// ---- POUs/HAWinoCore/MQTT.TcPOU
PROGRAM MQTT
VAR
// Local Variables for Mqtt Client handling
	fbIotMqttClient : FB_IotMqttClient;
	bSetParameter 	: BOOL := TRUE;
	bConnect 		: BOOL := TRUE;	
	
// Publish message
	initMQTT : BOOL := FALSE;
	sTopicPubToPowerMgmt : STRING(255); //:= CONCAT('Robots/PowerMgmt/Robot_', INT_TO_STRING(.Var_HAWIno.Robot_Number)); 	// ToDo: Bisher ist die Nummer des HAWino fest kodiert
	sTopicPubToPowerMgmt_SOC : STRING(255);// := CONCAT('Robots/PowerMgmt/SoC_Robot_', INT_TO_STRING(.Var_HAWIno.Robot_Number)); 
	sPayloadPub : STRING(2000);	
	fbTimerPub 	: TON := (PT:=T#500MS);									// Intervall für das Senden des Akku-Status
	
//Received message
	bSubscribed    : BOOL;
	sTopicSubToPowerMgmt : STRING(255);// := CONCAT('PowerMgmt/Robots/Robot_', INT_TO_STRING(.Var_HAWIno.Robot_Number));	// ToDo: Bisher ist die Nummer des HAWino fest kodiert
	sTopicRcv      : STRING(255);
	sPayloadRcv    : STRING(255);
	sPayloadRcv_Status    : STRING(255);
	sPayloadRcv_Status_Test: STRING(255);
	fbMessageQueue : FB_IotMqttMessageQueue;
    fbMessage      : FB_IotMqttMessage;
	hrErrorOccurred : HRESULT; 			// Enthlt dern letzten augetretenen Fehler
	
//subscribe
	sTopicSubToGW1_Status : STRING(255);
	sTopicSubToGW1_Auftrag : STRING(255);
	sTopicSubCollision : STRING(255);
	sTopicPubCollision : ARRAY[1..4] OF STRING(255);
	sTopicSubReset : STRING(255);
	
// Variables for JSON
	fbJson			: FB_JsonSaxWriter;
	fbJsonDataType 	: FB_JsonReadWriteDataType;
	sJsonDoc       	: STRING(2000); 
	
// Local Variables for TwinCAT IoT Communication (TF6701) with direct link to EK1200 and TcCom
	//stMqtt_HAWino_In	AT%I*	: ST_PwrMgmt_HAWino_In;		// Attention! Don't link TIME Variables, otherwise we get an error!
	//stMqtt_HAWino_Out	AT%Q*	: ST_PwrMgmt_HAWino_Out;
	
	stMqtt_HAWino_In	 AT%I*: ST_PwrMgmt_HAWino_In;		// Attention! Don't link TIME Variables, otherwise we get an error!
	stMqtt_HAWino_Out	 AT%Q*: ST_PwrMgmt_HAWino_Out;
	
	SOC_Out : STRING(255);
	nBatteryTemperature	AT%I*	: INT;
	
	bComCheckAnswer	AT%Q*	: BOOL;
	
	stMqtt_HAWinoValues	: ST_PwrMgmt_HAWino;
	
	
// Timer to create a time stamp
	fbTimerTimestamp : TON := (PT:=T#71582M47S295MS);
	
// Local Vaiables to evaluate and act to input
	fbComCheckFlag	: RS;
	
	sTopicSubToFleetMgmt: STRING;
	Reset1: BOOL;
	//Input synccheck. robotdata has been read and can be used.
	txtReadInit AT%I* : BOOL := FALSE;
	
	//eigene Topics und Payload
	sTopicPubToGW1 : STRING(255);
	WerkstueckAusgelesen: BOOL;
	sPayloadPub1 : STRING(2000);
	Robotstatus : RobotStatusGW1;
	sTopicSubToGW1: STRING(255);
	nPayloadSize:INT;
	sPayloadPubCollision : STRING(100);
	n: INT;												
	
	FeedbackToGW1 AT%I*: STRING(50);				//Statusmeldungen an Gewerk 1
	RoboNmbToGoBack AT%I* : ARRAY[0..4] OF INT;		//Nummer, der Roboter, die zurück sollen
	resetVar, resetGoBack AT%I*: BOOL;				//Reset Variablen, um Ausgänge zurückzusetzen
	Auftrag AT%Q*: Auftrag;							//Auftrag von Gewerk 1 gesendet
	StatusFromGW1 AT%Q*: STRING(50);				//Statusrückmeldungen von Gewerk 1 gesendet
	goBack AT%Q* : BOOL;							//true, wenn Roboter Platz machen soll
	resetButton AT%Q* : BOOL;						//Reset von Gewerk 1 kommend
END_VAR

//Case machen! preop op

//Unsere Topics und erwartete Struktur:
//Auftrag: {"Art":"Fahrauftrag","AbholStation":1,"AbholTasche":2,"AblageStation":3,"AblageTasche":1}
//Status: {"Status":"WerkstueckAusgelesen"}
//Kollision: {"todo":"goBack"}

IF txtReadInit THEN
	IF NOT initMQTT THEN
		sTopicPubToPowerMgmt  := CONCAT('Robots/PowerMgmt/Robot_', INT_TO_STRING(.Var_HAWIno.Robot_Number)); 	
		sTopicPubToPowerMgmt_SOC  := CONCAT('Robots/PowerMgmt/SoC_Robot_', INT_TO_STRING(.Var_HAWIno.Robot_Number)); 
		sTopicSubToPowerMgmt  := CONCAT('PowerMgmt/Robots/Robot_', INT_TO_STRING(.Var_HAWIno.Robot_Number));
		sTopicSubToGW1  := CONCAT('VPJ/Robot_', INT_TO_STRING(.Var_HAWIno.Robot_Number));
		sTopicSubToGW1_Status  := CONCAT(sTopicSubToGW1, '/Status');
		sTopicSubToGW1_Auftrag  := CONCAT(sTopicSubToGW1, '/Auftrag');
		sTopicPubToGW1 := CONCAT('VPJ/Robot_', INT_TO_STRING(.Var_HAWIno.Robot_Number));
		sTopicSubCollision := CONCAT('VPJ/Robot_', INT_TO_STRING(.Var_HAWIno.Robot_Number));
		sTopicSubCollision := CONCAT(sTopicSubCollision, '/Collision');
		sTopicSubReset  := CONCAT('VPJ/Robot_', INT_TO_STRING(.Var_HAWIno.Robot_Number));
		sTopicSubReset  := CONCAT(sTopicSubToGW1, '/Reset');
		FOR n := 1 TO 4 BY 1 DO
			IF n <> .Var_HAWIno.Robot_Number THEN
				sTopicPubCollision[n] := CONCAT('VPJ/Robot_', INT_TO_STRING(n));
				sTopicPubCollision[n] := CONCAT(sTopicPubCollision[n], '/Collision');
			END_IF
		END_FOR
		initMQTT:= TRUE;
	END_IF
	
	stMqtt_HAWinoValues.Output.nRobotNumber := .Var_HAWIno.Robot_Number;			// Anpassen für jeden HAWino
	
	fbTimerTimestamp(In:= NOT fbTimerTimestamp.Q, ET=>stMqtt_HAWinoValues.Output.tTimestamp);
	
	stMqtt_HAWinoValues.Output.fSoC := stMqtt_HAWino_In.fSoC;
	
	stMqtt_HAWinoValues.Output.fActualBatteryCurrent := stMqtt_HAWino_In.fActualBatteryCurrent;
	stMqtt_HAWinoValues.Output.fActualBatteryVoltage := stMqtt_HAWino_In.fActualBatteryVoltage;

	
	// Skalierung der Temperaturwerte des Akkus
	stMqtt_HAWinoValues.Output.fBatteryTemperature := FKT_Scale(Rohwert := nBatteryTemperature, 
																	X1 := -500,
																	X2 := 1500, 
																	Y1 := -50,
																	Y2 := 150);
																	
	// Ausgabe der erwarteten Laufzeit des Roboters
	stMqtt_HAWinoValues.Output.nEstimatedRunningTime	:= LIMIT(0,stMqtt_HAWino_In.nEstimatedRunningTime,172800);		// Max. 48 Stunden sollen dargestellt werden
	stMqtt_HAWinoValues.Output.nEstimatedChargingTime	:= LIMIT(0,stMqtt_HAWino_In.nEstimatedChargingTime,172800);		// Max. 48 Stunden sollen dargestellt werden
	
	
	// Antworten auf den Kommunikationstest und des Ladetests
	stMqtt_HAWinoValues.Output.bCheckCurrentDetected := stMqtt_HAWino_In.bCheckCurrentDetected;
	stMqtt_HAWinoValues.Output.bComCheckAnswer := stMqtt_HAWino_In.bComCheckAnswer;
	
	//
	// Setting the parameters for establishing the connection to the Mqtt Broker and initializing the connection.
	//
	IF bSetParameter THEN
		fbIotMqttClient.sHostName := '192.168.0.11';	// IP-Adresse des Servers
		fbIotMqttClient.nHostPort := 1883;
		//fbIotMqttClient.sClientId := ClientId;
		fbIotMqttClient.sClientId := CONCAT('Robot_', INT_TO_STRING(.Var_HAWIno.Robot_Number));
		fbIotMqttClient.sTopicPrefix := '';
		//fbIotMqttClient.nKeepAlive:= 60; 
		fbIotMqttClient.sUserName:= 'VPJ';
		fbIotMqttClient.sUserPassword:= 'R462';
		//fbIotMqttClient.stWill:= ; 
		//fbIotMqttClient.stTLS:= ;
		fbIotMqttClient.ipMessageQueue := fbMessageQueue;
	
		bSetParameter := FALSE;
	END_IF
	
	
	//
	// This method -> MUST BE CALLED CYCLICALLY <- to ensure background communication with the MQTT broker.
	//
	fbIotMqttClient.Execute(bConnect);
	
	IF fbIotMqttClient.bError THEN
		// ToDo: add error logging here
		hrErrorOccurred := fbIotMqttClient.hrErrorCode;
	END_IF
	
		
	IF fbIotMqttClient.bConnected THEN		// Kontrolle, ob der Broker verbunden ist
		IF NOT bSubscribed THEN
			//
			// Abbonieren der Toopics, welche vom PowerMgmt kommen
			//
			bSubscribed := fbIotMqttClient.Subscribe(sTopic:=sTopicSubToPowerMgmt, eQoS:=TcIotMqttQos.AtMostOnceDelivery);
			IF fbIotMqttClient.bError THEN
				// ToDo: add my error logging here
				hrErrorOccurred := fbIotMqttClient.hrErrorCode;
			END_IF
			
			//
			// Abbonieren der Toopics, welche vom Gewerk 1 kommen
			//
			//Abbonieren von Topics: VPJ/Roboter
			bSubscribed := fbIotMqttClient.Subscribe(sTopic:=sTopicSubToGW1_Status, eQoS:=TcIotMqttQos.AtMostOnceDelivery);
			bSubscribed := fbIotMqttClient.Subscribe(sTopic:=sTopicSubToGW1_Auftrag, eQoS:=TcIotMqttQos.AtMostOnceDelivery);
			bSubscribed := fbIotMqttClient.Subscribe(sTopic:=sTopicSubCollision, eQoS:=TcIotMqttQos.AtMostOnceDelivery);
			bSubscribed := fbIotMqttClient.Subscribe(sTopic:=sTopicSubReset, eQoS:=TcIotMqttQos.AtMostOnceDelivery);
			
			
			//bSubscribed := fbIotMqttClient.Subscribe(sTopic:=sTopicSubToFleetMgmt, eQoS:=TcIotMqttQos.AtMostOnceDelivery);
			//IF fbIotMqttClient.bError THEN
				// ToDo: add my error logging here
			//	hrErrorOccurred := fbIotMqttClient.hrErrorCode;
			//END_IF
			
		END_IF
	END_IF	
	
	
	
	// Senden der MQTT- Nachrichten
	
	
	IF fbIotMqttClient.bConnected THEN			// Kontrolle, ob Broker verbunden ist
		fbTimerPub(IN:=TRUE);
		
		//
		// publish new paylod every 500 MS
		//
		IF fbTimerPub.Q THEN					// Abwarten des oben eingestellten Intervalls
			fbTimerPub(IN:=FALSE);
			
			//
			// Nachricht an PowerMgmt
			//
			fbJson.ResetDocument();
			fbJsonDataType.AddJsonValueFromSymbol(fbJson, 'ST_PwrMgmt_HAWino_In', SIZEOF(stMqtt_HAWinoValues.Output), ADR(stMqtt_HAWinoValues.Output));
			//sJsonDoc := fbJson.GetDocument();
			fbJson.CopyDocument(sJsonDoc, SIZEOF(sJsonDoc));
			
			sPayloadPub := sJsonDoc;	
			fbIotMqttClient.Publish(sTopic:= sTopicPubToPowerMgmt, 
										pPayload:= ADR(sPayloadPub), 
										nPayloadSize:= LEN2(ADR(sPayloadPub))+1, 										
										eQoS:= TcIotMqttQos.AtMostOnceDelivery, 
										bRetain:= FALSE, 
										bQueue:= FALSE);
									
									
			
			SOC_Out	:= CONCAT( '{"SoC" : ',LREAL_TO_STRING(stMqtt_HAWinoValues.Output.fSoC));
			SOC_Out	:= CONCAT( SOC_Out,'}');
			
			
			
			
			//SOC_Out := 	LREAL_TO_STRING(stMqtt_HAWinoValues.Output.fSoC);
			
						
			fbIotMqttClient.Publish(sTopic:= sTopicPubToPowerMgmt_SOC, 
										pPayload:=ADR(SOC_Out), 
										nPayloadSize:= INT_TO_UDINT(LEN(SOC_Out)),
										eQoS:= TcIotMqttQos.AtMostOnceDelivery, 
										bRetain:= FALSE, 
										bQueue:= FALSE);
										
										
			IF fbIotMqttClient.bError THEN
				// ToDo: add error logging here
				hrErrorOccurred := fbIotMqttClient.hrErrorCode;
			END_IF	
			
			//
			// Nachricht an GW1 - Produktionsauftrag
			//
			
			//Rückmeldung Roboterstatus
			sPayloadPub1 := CONCAT( '{"Status" : ', FeedbackToGW1);
			sPayloadPub1 := CONCAT( sPayloadPub1,'}');
			
			fbIotMqttClient.Publish(sTopic:= sTopicPubToGW1, 
											pPayload:=ADR(sPayloadPub1), 
											nPayloadSize:= INT_TO_UDINT(LEN(sPayloadPub1)),
											eQoS:= TcIotMqttQos.AtMostOnceDelivery, 
											bRetain:= FALSE, 
											bQueue:= FALSE);
											
			//An alle Roboter, die an Kollision beteiligt sind, goBack senden
			FOR n := 0 TO 4 BY 1 DO
				IF RoboNmbToGoBack[n] > 0 THEN
					sPayloadPubCollision := '{"todo":"goBack"}';
					
					fbIotMqttClient.Publish(sTopic:= sTopicPubCollision[RoboNmbToGoBack[n]], 
													pPayload:=ADR(sPayloadPubCollision), 
													nPayloadSize:= INT_TO_UDINT(LEN(sPayloadPubCollision)),
													eQoS:= TcIotMqttQos.AtMostOnceDelivery, 
													bRetain:= FALSE, 
													bQueue:= FALSE);
				END_IF
			END_FOR
		END_IF
	END_IF
	
	
	// Verarbeiten der Subscriptions
	
	
	IF fbMessageQueue.nQueuedMessages > 0 THEN			// Kontrolle, ob neue Daten vorliegen
		IF fbMessageQueue.Dequeue(fbMessage:=fbMessage) THEN
			fbMessage.GetTopic(pTopic:=ADR(sTopicRcv), nTopicSize:=SIZEOF(sTopicRcv) );
			

				
			//
			// Message from PowerMgmt
			//
			IF fbMessage.CompareTopic(sTopic:=sTopicSubToPowerMgmt) THEN		// Wenn die Daten vom PowerMgmt kommen, dann führe folgenede Aktion aus
				fbMessage.GetPayload(pPayload:=ADR(sPayloadRcv), nPayloadSize:=SIZEOF(sPayloadRcv), bSetNullTermination:=FALSE);
			// Json-String aufteilen und in Variablen schreiben
				fbJsonDataType.SetSymbolFromJson(sPayloadRcv,'ST_PwrMgmt_HAWino_Out',SIZEOF(stMqtt_HAWinoValues.Input),ADR(stMqtt_HAWinoValues.Input));
			END_IF
		
			//
			// Hier werden weitere Topics verarbeitet
			// 
			//Status von Gewerk 1 kommend
			IF fbMessage.CompareTopic(sTopic:=sTopicSubToGW1_Status) THEN
				
				fbMessage.GetPayload(pPayload:=ADR(sPayloadRcv_Status), nPayloadSize:=SIZEOF(sPayloadRcv_Status), bSetNullTermination:=true);
				// Json-String aufteilen und in Variablen schreiben
				fbJsonDataType.SetSymbolFromJson(sPayloadRcv_Status,'RobotStatusGW1',SIZEOF(RobotStatus),ADR(RobotStatus));
				StatusFromGW1 := Robotstatus.Status;
				Robotstatus.Status := '';
				sPayloadRcv_Status := '';
			END_IF
			
			//Auftrag von Gewerk 1 kommend
			IF fbMessage.CompareTopic(sTopic:=sTopicSubToGW1_Auftrag) THEN
				fbMessage.GetPayload(pPayload:=ADR(sPayloadRcv), nPayloadSize:=SIZEOF(sPayloadRcv), bSetNullTermination:=TRUE);
			
			// Json-String aufteilen und in Variablen schreiben
				fbJsonDataType.SetSymbolFromJson(sPayloadRcv,'Auftrag',SIZEOF(Auftrag),ADR(Auftrag));
			END_IF
			
			//Nachricht von anderem HAWino, dass dieser zurückfahren soll
			IF fbMessage.CompareTopic(sTopic:=sTopicSubCollision) THEN
				goBack := TRUE;
			END_IF
			
			//Nachricht von Gewerk 1, dass HAWino reset machen soll (nach Fehler)
			IF fbMessage.CompareTopic(sTopic:=sTopicSubReset) THEN
				resetButton := TRUE;
			END_IF
			
		END_IF
	END_IF	
	
	//Rücksetzen der durch Gewerk 1 beschriebenen Variablen
	IF resetVar THEN
		StatusFromGW1 := '';
		Robotstatus.Status := '';
		sPayloadRcv_Status := '';
		Auftrag.AbholStation := 0;
		Auftrag.AbholTasche := 0;
		Auftrag.AblageStation := 0;
		Auftrag.AblageTasche := 0;
		Auftrag.Art := '';
		resetButton := FALSE;
	END_IF
	
	IF resetGoBack THEN
		goBack := FALSE;
	END_IF
	
	
	// Evaulierung der empfangenen Daten
	
	//
	// ToDo: Plausibilitätsprüfung von stMqtt_HAWinoValues.Input und evt. TypConversion
	// Attention! The assignment of input to output is correct. Don `t change!
	//	
	
	stMqtt_HAWino_Out.bChargingActive := stMqtt_HAWinoValues.Input.bChargingActive;
	stMqtt_HAWino_Out.bExternalRecalibrationTrigger := stMqtt_HAWinoValues.Input.bExternalRecalibrationTrigger;
	stMqtt_HAWino_Out.fExternalRecalibrationValue := stMqtt_HAWinoValues.Input.fExternalRecalibrationValue;
	
	
	// Hier Communication Check einbauen
	
	//fbComCheckFlag(Set:= stMqtt_HAWinoValues.Input.bComCheckRequest, 
	//					Reset1:= NOT stMqtt_HAWinoValues.Input.bComCheckRequest,
	//					Q1 => bComCheckAnswer);
	bComCheckAnswer	:= TRUE;
					
END_IF

END_PROGRAM

// ---- POUs/UserPOUs/FKT_Scale.TcPOU
FUNCTION FKT_Scale : LREAL
VAR_INPUT
	// Unterer Auflösungsbereich
	X1: LREAL;
	// Oberer Auflösungsbereich
	X2: LREAL;
	// Unterer Darstellungsbereich
	Y1: LREAL;
	// Oberer Darstellungsbereich
	Y2: LREAL;
END_VAR
VAR
	// Rohwert in Real
	X: LREAL;
	// Skalierter Messwert
	Y: LREAL := 0;
END_VAR
VAR_INPUT
	// Analoger Eingang in 12 bzw. 16 Bit
	Rohwert: LREAL;
END_VAR

X := Rohwert;

Y := ((((Y2-Y1)/(X2-X1))*(X-X1))+Y1);			// Skalierung über eine lineare Funktion

IF Y > Y2 THEN
	Y := Y2;									// Obere Begrenzung
ELSIF Y < Y1 THEN
	Y := Y1;									// Untere Begrenzung
END_IF

FKT_Scale := Y;									// Ausgabe

END_FUNCTION

// ---- POUs/HAWinoCore/HAWino.TcPOU
PROGRAM HAWino
VAR
	//CX35CDD6
	Robot_Number	AT%Q*	: INT;
	operationState : DUT_SysState := DUT_SysState.init; 
	RobotData : RobotInternalData;
	GetId : Tc2_Utilities.FB_GetSystemId;
	init : INT;
	SysGUID : GUID;
	start : BOOL:= TRUE;
	initDone AT%Q* : BOOL := FALSE;
END_VAR

CASE operationState OF
	//Get SysId for Identification
	DUT_SysState.init:
		GetId(bexecute := start,stSystemId=>SysGUID);
		IF NOT GetId.bBusy THEN	
			operationState:=DUT_SysState.preOp;
		END_IF
	DUT_SysState.preOp:
	//Set RobotNumber for MQTT and set flag to start MQTT
		IF InitSysId(GUID_to_String(SysGUID)) THEN
			Var_HAWIno.Robot_Number := RobotData.Robot_Number;		
			initDone := TRUE;
			operationState:=DUT_SysState.Op;
		END_IF
	DUT_SysState.Op:
	//Operate System
		//MotorDrivers();
		//WheelEncoders();
		IrDistanceSensors();
		Camera();
		PowerManager();
		Gripper();
		
END_CASE

METHOD InitSysId : BOOL
VAR_INPUT
	SysId : STRING;
END_VAR
VAR
	state : INT;
	CX31C9D6 : STRING := '77726FC0-DD5E-F7D7-002E-41ED9B95AABA';
	CX35CFB8 : STRING := '2A7FC16A-555A-D05D-0E28-E804E05477FE';
	CX35CDC8 : STRING := 'AD3D576A-9CE4-FB95-7439-909C21AA2B33';
	CX35CDD6 : STRING := '975A6B25-37E2-0E46-4C4D-43CCC26F2A66';
	CX4D0046 : STRING := '4FFA7061-8E1F-E1C9-731A-38EAA9BAEAC6';
END_VAR
// CX-31C9D6 = 1
// CX-35CFB8 = 2
// CX-35CDC8 = 3
// CX-35CDD6 = 4
// CX-4D0046 = 5
IF SysId = CX31C9D6 THEN
	state := 1;
ELSIF SysId = CX35CFB8 THEN
	state := 2;
ELSIF SysId = CX35CDC8 THEN
	state := 3;
ELSIF SysId = CX35CDD6 THEN
	state := 4;
ELSIF SysId = CX4D0046 THEN
	state := 5;
ELSE
	state := 0;
END_IF

CASE state OF 
		1 : 	
				RobotData.Robot_IP_WiFi :='192.169.0.18';
				RobotData.Robot_IP_Wire :='192.169.0.28';
				RobotData.Robot_Name :='CX-35C9D6';
				RobotData.Robot_Nickname :='9D6';
				RobotData.Robot_Number := 1;
				InitSysId := True;
		2:
				RobotData.Robot_IP_WiFi :='192.169.0.17';
				RobotData.Robot_IP_Wire :='192.169.0.27';
				RobotData.Robot_Name :='CX-35CFB8';
				RobotData.Robot_Nickname :='FB8';
				RobotData.Robot_Number := 2;
				InitSysId := TRUE;
		3:
				RobotData.Robot_IP_WiFi :='192.169.0.16';
				RobotData.Robot_IP_Wire :='192.169.0.26';
				RobotData.Robot_Name :='CX-35CDC8';
				RobotData.Robot_Nickname :='DC8';
				RobotData.Robot_Number := 3;
				InitSysId := TRUE;
		4:
				RobotData.Robot_IP_WiFi :='192.169.0.15';
				RobotData.Robot_IP_Wire :='192.169.0.25';
				RobotData.Robot_Name :='CX-35CDD6';
				RobotData.Robot_Nickname :='DD6';
				RobotData.Robot_Number := 4;
				InitSysId := TRUE;
		5:
				RobotData.Robot_IP_WiFi :='192.169.0.19';
				RobotData.Robot_IP_Wire :='192.169.0.29';
				RobotData.Robot_Name :='CX-04D0046';
				RobotData.Robot_Nickname :='046';
				RobotData.Robot_Number := 5;
				InitSysId := TRUE;			
		ELSE	//Ungültige Roboter Nummer
				RobotData.Robot_IP_WiFi :='0.0.0.0';
				RobotData.Robot_IP_Wire :='0.0.0.0';
				RobotData.Robot_Name :='Invalid';
				RobotData.Robot_Nickname :='Invalid';
				RobotData.Robot_Number := 0;
				InitSysId := false;
	END_CASE;
END_METHOD

END_PROGRAM

// ---- POUs/HAWinoCore/IrDistanceSensors.TcPOU
PROGRAM IrDistanceSensors
VAR
	distanceRaw AT %I* : ARRAY [1..9] OF INT;
	
	distance_mm AT %Q* : ARRAY [1..9] OF REAL;

	i : INT;
END_VAR

FOR  i := 1 TO 9 DO
	distance_mm[i] := IrDistanceFromRaw(distanceRaw[i]);
END_FOR

END_PROGRAM

// ---- POUs/HAWinoCore/IrDistanceFromRaw.TcPOU
FUNCTION IrDistanceFromRaw : REAL
VAR_INPUT
	rawValue : INT;
END_VAR
VAR
END_VAR

	IrDistanceFromRaw := 123.15 / EXPT( INT_TO_REAL(rawValue) * (10.0 / 32767.0), 1.119 );

END_FUNCTION

// ---- POUs/HAWinoCore/Camera.TcPOU
PROGRAM Camera
VAR
		cameraData : CameraConnectionUDP;
END_VAR

cameraData();

END_PROGRAM

// ---- POUs/HAWinoCore/CameraConnectionUDP.TcPOU
{attribute 'c++_compatible'}
FUNCTION_BLOCK CameraConnectionUDP IMPLEMENTS ITcIoUdpProtocolRecv
VAR_INPUT
END_VAR
VAR_OUTPUT
	robotPositionArray : ARRAY [1..8] OF RobotPose; 
END_VAR
VAR
	{attribute 'TcInitSymbol'}
	oid : OTCID; // To be set in PLC_Instance object and required for FW_ObjMgr_GetObjectInstance()
	ipUdp : ITcIoUdpProtocol;
	nUdpPort : UINT := 25000;
	nReceivedPakets : UINT;
	//uLastReceivedIP : U_IpAdr; 
	hrInit : HRESULT;
	hrSend  : HRESULT; 
	robotPosition AT %Q* : ARRAY [1..8] OF RobotPose; 
	
	HH					AT	%Q*	:	LREAL;	
	MM					AT	%Q*	:	LREAL;
	SS					AT	%Q*	:	LREAL;
	
	counter	:	UDINT	:= 0;
	x1,y1,theta1,x2,y2,theta2,x3,y3,theta3,x4,y4,theta4,x5,y5,theta5 : LREAL;
END_VAR


IF ipUdp <> 0 THEN
	ipUdp.CheckReceived();
END_IF



x1 := robotPosition[1].x;
y1 := robotPosition[1].y;
theta1 := robotPosition[1].theta;
x2 := robotPosition[2].x;
y2 := robotPosition[2].y;
theta2 := robotPosition[2].theta;
x3 := robotPosition[3].x;
y3 := robotPosition[3].y;
theta3 := robotPosition[3].theta;
x4 := robotPosition[4].x;
y4 := robotPosition[4].y;
theta4 := robotPosition[4].theta;
x5 := robotPosition[5].x;
y5 := robotPosition[5].y;
theta5 := robotPosition[5].theta;

robotPositionArray := robotPosition;

{attribute 'conditionalshow'}
METHOD FB_exit : BOOL
VAR_INPUT
	bInCopyCode : BOOL; // if TRUE, the exit method is called for exiting an instance that is copied afterwards (online change).
END_VAR
IF NOT bInCopyCode THEN // no online change
	IF ipUdp <> 0 THEN 
		ipUdp.UnregisterReceiver(nUdpPort); // Shutdown
		FW_SafeRelease(ADR(ipUdp));
		FB_exit := TRUE; 
	END_IF
END_IF
END_METHOD

{attribute 'conditionalshow'}
METHOD FB_init : BOOL
VAR_INPUT
	bInitRetains : BOOL; // if TRUE, the retain variables are initialized (warm start / cold start)
	bInCopyCode : BOOL;  // if TRUE, the instance afterwards gets moved into the copy code (online change)
END_VAR
VAR
	ipSrv : ITComObjectServer;
END_VAR
IF NOT bInCopyCode THEN // no online change
	IF ipUdp = 0 THEN
	    hrInit := FW_ObjMgr_GetObjectInstance(	oid:=oid, 
											iid:=TC_GLOBAL_IID_LIST.IID_ITcIoUdpProtocol, 
											pipUnk:=ADR(ipUdp) );
		IF SUCCEEDED(hrInit) THEN 
			IF  SUCCEEDED(ipUdp.RegisterReceiver(nUdpPort, THIS^)) THEN //open port
				FB_init := TRUE;
			ELSE 
				FW_SafeRelease(ADR(ipUdp));
			END_IF
		END_IF				
	END_IF
END_IF
END_METHOD

{attribute 'conditionalshow'}
METHOD FB_reinit : BOOL
VAR_INPUT
END_VAR
IF (ipUdp <> 0) THEN 
	ipUdp.RegisterReceiver(nUdpPort, THIS^);
	FB_reinit := TRUE; 
END_IF
END_METHOD

{attribute 'object_name' := 'ReceiveData'}
{attribute 'c++_compatible'}
{attribute 'signature_flag' := '33554688'}
{attribute 'pack_mode' := '4'}
{attribute 'show'}
{attribute 'minimal_input_size' := '4'}
METHOD ReceiveData : HRESULT
VAR_INPUT
	ipAddr	: UDINT;
	udpDestPort	: UINT;
	udpSrcPort	: UINT;
	nData	: UDINT;
	pData	: PVOID;
	pVlan	: POINTER TO ETYPE_VLAN_HEADER := 0;
END_VAR
VAR 
	i : INT;
	x,y,theta,e : LREAL;
	hou, minu, sek : LREAL;
	DataUDP : STRING;
END_VAR
nReceivedPakets := nReceivedPakets+1;
//uLastReceivedIP.ipAdrInternal := ipAddr;


	(*** Auslesen des Datenbereichs von UDP-Paketen ***
	* UDP-Telegramm besteht aus 56*8 = 448 Bytes (siehe UDP-Doku Lokalisierungsrechner)
	  Pro Robotino: 3*8 = 24 Bytes: je 8 Bytes für x-Koord, y-Koord, theta in rad
	  Robotino1: Bytes 1-8   -> x-Koord, Bytes 9-16  -> y-Koord, Bytes 17-24 -> theta
	  Robotino2: Bytes 25-32 -> x-Koord, Bytes 33-40 -> y-Koord, Bytes 41-48 -> theta  usw.. 
	* pData zeigt auf Adressbereich, in dem die 448 Byte großen UDP-Daten liegen
	  in der Schleife werden jeweils 8 Byte in den UDP-Array geschrieben und der Pointer nach
	  jedem Schritt um 8 Byte weiter geschoben.*)
	
IF nData = 448 THEN

	FOR i := 1 TO 8 DO
		memcpy( ADR(x), 	pData + 8 * 0 + 4*8*(i-1), 8);			// x-Koord
		memcpy( ADR(y),    	pData + 8 * 1 + 4*8*(i-1), 8);			// y-Koord
		memcpy( ADR(theta), pData + 8 * 2 + 4*8*(i-1), 8);			// theta
		memcpy( ADR(e), 	pData + 8 * 3 + 4*8*(i-1), 8);			// e
		
		robotPosition[i].x  := (x);
		robotPosition[i].y := (y);
		robotPosition[i].theta := (theta);
		robotPosition[i].e := (e);
			
	END_FOR
	memcpy( ADR(HH), pData + 256, 8);						// Hours
	memcpy( ADR(MM), pData + 264, 8);						// Minutes
	memcpy( ADR(SS), pData + 272, 8);						// Seconds
//	memcpy( ADR(hou), pData + 64, 8);						// Hours
//	memcpy( ADR(minu), pData + 200, 8);						// Minutes
//	memcpy( ADR(sek), pData + 208, 8);						// Seconds
	
//	HH := (hou);
//	MM := (minu);
//	SS := (sek);

//	DataUDP := pData^;

END_IF
END_METHOD

{attribute 'object_name' := 'TcAddRef'}
{attribute 'c++_compatible'}
{attribute 'signature_flag' := '33554688'}
{attribute 'pack_mode' := '4'}
{attribute 'show'}
{attribute 'minimal_input_size' := '4'}
METHOD TcAddRef : UDINT
END_METHOD

{attribute 'object_name' := 'TcQueryInterface'}
{attribute 'c++_compatible'}
{attribute 'signature_flag' := '33554688'}
{attribute 'pack_mode' := '4'}
{attribute 'show'}
{attribute 'minimal_input_size' := '4'}
METHOD TcQueryInterface : HRESULT
VAR_INPUT
	iid	: REFERENCE TO IID;
	pipItf	: POINTER TO PVOID;
END_VAR
VAR
	ipUdpRecv : ITcIoUdpProtocolRecv;
	ipUnknown : ITcUnknown;	
END_VAR
IF GuidsEqual(ADR(iid), ADR(TC_GLOBAL_IID_LIST.IID_ITcIoUdpProtocolRecv)) THEN
	ipUdpRecv := THIS^; // cast to interface pointer
	pipItf^ := ITCUNKNOWN_TO_PVOID(ipUdpRecv);
	TcAddRef();
	TcQueryInterface := S_OK;
ELSIF GuidsEqual(ADR(iid), ADR(TC_GLOBAL_IID_LIST.IID_ITcUnknown)) THEN
	ipUnknown := THIS^; // cast to interface pointer
	pipItf^ := ITCUNKNOWN_TO_PVOID(ipUnknown);
	TcAddRef();
	TcQueryInterface := S_OK;
ELSE
	TcQueryInterface := E_HRESULTAdsErr.NOINTERFACE ; //Call super if this fb extends some other
END_IF
END_METHOD

{attribute 'object_name' := 'TcRelease'}
{attribute 'c++_compatible'}
{attribute 'signature_flag' := '33554688'}
{attribute 'pack_mode' := '4'}
{attribute 'show'}
{attribute 'minimal_input_size' := '4'}
METHOD TcRelease : UDINT
END_METHOD

END_FUNCTION_BLOCK

// ---- POUs/HAWinoCore/PowerManager.TcPOU
PROGRAM PowerManager
VAR
	shutdownButton			AT%I*  : BOOL := FALSE;
	batteryVoltageRaw  		AT%I*  : INT;
	shutdownTrigger 		AT%Q*  : BOOL := FALSE;
	batteryVoltage_V		AT%Q*  : REAL;
	
	supplyCurrentRaw		AT%I* : INT;
	supplyCurrent_A			AT%Q* : REAL; 
	
	SOC AT%I* : REAL;
	
	requestShutdown 		AT%I* : BOOL;
	
	shutdown: NT_Shutdown;

	scaleVoltage:	REAL := LREAL_TO_REAL(20/EXPT(2,16)); 		// (Spannungsbereich der Klemme)/(Wertebereich)
	dummy:  REAL;
	
	stMqtt_HAWino_IN	AT%Q*	: ST_PwrMgmt_HAWino_In;			// Link MQTT-DatenStruct
	
	shut: INT;
END_VAR

IF shutdownButton THEN
	shutdown(DELAY:=1, START:=TRUE);
END_IF

batteryVoltage_V := (batteryVoltageRaw * scaleVoltage * 2.0);

//batteryVoltage_V := batteryVoltageRaw;

supplyCurrent_A :=  supplyCurrentRaw * 1000.0 / 270.0 / 32768 * 10;
//supplyCurrent_A :=  supplyCurrentRaw;
// TODO: Filter and CALIBRATE this!
//shutdownTrigger := requestShutdown ;// OR batteryVoltage_V < 14.0;

IF batteryVoltage_V < 12 AND SOC < 10 THEN
	
	//shutdownTrigger := TRUE;

END_IF

stMqtt_HAWino_IN.fActualBatteryVoltage := batteryVoltage_V;
stMqtt_HAWino_IN.fActualBatteryCurrent := supplyCurrent_A;


//stMqtt_HAWino_In.fActualBatteryVoltage := batteryVoltage_V;
//stMqtt_HAWino_In.fActualBatteryCurrent := supplyCurrent_A

END_PROGRAM

// ---- POUs/HAWinoCore/Gripper.TcPOU
PROGRAM Gripper
VAR_INPUT
END_VAR
VAR
	closeGripperFromSimulink AT%I* : LREAL:=0;
	closeGripperCommand		AT%I* : BOOL;					//True: opening, false: closing
	slider					AT%I* : BOOL;
	partGripped				AT%I* : BOOL;					//Teil zwischen Greifer: partGripped := 0
	
	sliderToSimulink 		AT%Q* : LREAL:=0;
	partInGripperToSimulink AT%Q*  :LREAL:=0;
	
	driveEnable				AT%Q* : BOOL;
	driveVelocity 			AT%Q* : INT;
	
	state : CoreGripperControlState := CoreGripperControlState.Closed;	//bei open hat der Greifer gegriffen (war mit open initialisiert)
	
	timer : TON;
	
	movementTime : TIME := T#1.0S;
	
END_VAR

CASE state OF 
		
	CoreGripperControlState.Opening:
		driveEnable:=1;
		driveVelocity:=-32767;
		timer(IN:=1);
		
		IF timer.Q THEN state := CoreGripperControlState.Open;
		END_IF
		
		IF closeGripperFromSimulink < 0.5 AND NOT closeGripperCommand THEN
			state := CoreGripperControlState.Closing;
			timer(in := 0, pt:= movementTime);
		END_IF
		
	CoreGripperControlState.Closing:
		driveEnable:=1;
		driveVelocity:=32767;
		timer(IN:=1);
		
		IF timer.Q THEN state := CoreGripperControlState.Closed;
		END_IF
		
		IF closeGripperFromSimulink > 0.5 OR  closeGripperCommand THEN
			state := CoreGripperControlState.Opening;
			timer(in := 0, pt:= movementTime);
		END_IF
		
		
	CoreGripperControlState.Open:	
		driveEnable:=0;
		driveVelocity:=0;

		IF closeGripperFromSimulink < 0.5 AND NOT closeGripperCommand THEN
			state := CoreGripperControlState.Closing;
			timer(in := 0, pt:= movementTime);
		END_IF
		
	CoreGripperControlState.Closed:	
		driveEnable:=0;
		driveVelocity:=0;
		
		IF closeGripperFromSimulink > 0.5 OR closeGripperCommand THEN
			state := CoreGripperControlState.Opening;
			timer(in := 0, pt:= movementTime);
		END_IF
		
END_CASE

sliderToSimulink:=BOOL_TO_LREAL(NOT(slider));
partInGripperToSimulink:=BOOL_TO_LREAL(NOT(partGripped));

END_PROGRAM

// ---- POUs/UserPOUs/GW2/Fahrauftrag.TcPOU
PROGRAM Fahrauftrag
VAR
	//States für Hauptprogramm und Kollision
	sStart : BOOL := TRUE;
	s0,s1a,s1b,s2,s3,s4,s5,s6a,s6b,s7,s8,s9,s10,s11a,s11b,s12,s13,s14,s15,s16,s17,s18,s19,s20,s21a,s21b,s22,s23,s24,s25,s25b,s26a,s26b,s27,s28,s29,s30,s31,s32,s33,s34,s35: BOOL := FALSE;
	sk0, sk1, sk2, sk3, sk4, sk10, sk20, sk21, sk22, sk23, sk24, sk25, sk26, sk27, sk28, sk29, sk30, sk31, sk32, sk33 : BOOL := FALSE; //States von Kollision
	
	AStar : AStar;										//A-Stern Algorithmus
	readAssigment: ReadAssigment;						//Auswertung des Auftrags
	TrajectoryController: TrajectoryControl;			//Schnittstelle zu GW3
	
	wayPointList : ARRAY[0..100] OF RobotPoseSimple;	//Wegpunktliste
	actualCamX, actualCamY : LREAL;						//letzte Kameradaten ungleich 0
	lastRelevantStateForCollision : STRING(5);			//letzter State für Rückfall bei Kollision
	
	//Schnittstelle zum MQTT_PRG
	FeedbackToGW1 AT%Q*: STRING(50);					//Feedback/Status des Roboters an GW1
	resetVarMQTT, resetGoBack AT%Q*: BOOL;				//messages von MQTT zurücksetzen
	RoboNmbToGoBack AT%Q* : ARRAY[0..4] OF INT;			//Roboter, die bei Kollision weichen sollen
	Auftrag AT%I*: Auftrag;								//Auftrag von GW1
	StatusFromGW1 AT%I*: STRING(50);					//Status von GW1
	goBack AT%I* : BOOL;								//zurückfahren auf Befehl von anderem HAWino
	reset AT%I* : BOOL;									//Fahrauftrag und GW3 zurücksetzen auf Befehl von GW1
	
	//Schnittstelle zu A*-Algorithmus
	EndNode : INT;							//letzter Knoten
	xEndvalue : LREAL;						//Ziel xKoordinate
	xRobotStartposition : LREAL;			//aktuelle xKoordinate
	yEndvalue : LREAL;						//Ziel yKoordinate
	yRobotStartposition : LREAL;			//aktuelle yKoordinate
	xPointList : ARRAY[0..100] OF LREAL;	//xKoordinatenliste
	yPointList : ARRAY[0..100] OF LREAL;	//yKoordinatenliste
	finished_ASearch : BOOL;	 			//Variable, dass Algorithmus fertig
	i: INT;									//Laufvariable zum Übertragen der x und y Koordinaten in die Wegpunktliste
	zeile: INT;								//Arrayindex, wo Wegpunktliste zuende
	
	//Kollision
	collision AT%I*: ARRAY[0..4] OF BOOL;				//Collision wurde erkannt
	lastCollision: ARRAY [0..4] OF BOOL;				//letzte Collision gespeichert
	collisionFree, collisionSolutionWorking : BOOL;		//keine Kollision aktuell
	removeNodeCollision : ARRAY[1..11] OF INT;			//Nodes die durch anderen HAWino blockiert
	todo : STRING(10);									//Aufgabe von diesem HAWino bei Kollision (fahren oder warten)
	firstTime: BOOL := TRUE;	
	timerCollision : TON;								//Zeit die bei Kollision gewartet wird, bevor Reaktion folgt
	otherRobo : ARRAY[0..4] OF INT;						//andere HAWinos, die an Kollision beteilgit
	otherRoboAtStation, otherRoboAtStop, thisRoboAtStation, drivingAtStation, newCollision, sameStation : BOOL;
	
	//Greifer
	closeGripperCommand AT%Q* : BOOL;	
	
	//error
	noCamera, error : BOOL;
	resetTimer : TON;
	failedCounter: INT;
	cameraX, cameraY : ARRAY[1..4] OF LREAL;
END_VAR

timerCollision();
resetTimer();
errorTest();
CameraDataSaved();

////////////////////////////////////////////////////////////Kollisionsauswertung///////////////////////////////////////////////////

collisionFree := NOT collision[Var_HAWIno.Robot_Number];

IF lastCollision[1] <> collision[1] OR lastCollision[2] <> collision[2] OR lastCollision[3] <> collision[3] OR lastCollision[4] <> collision[4] OR collision[0] THEN
	IF collision[Var_HAWIno.Robot_Number] THEN
		newCollision := TRUE;
	END_IF
	lastCollision := collision;
END_IF

IF collision[Var_HAWIno.Robot_Number] AND newCollision AND NOT collisionSolutionWorking THEN
	TrajectoryController.xBoEnable := FALSE;
	sk0 := TRUE;
	CollisionsSolution_new();
	newCollision := FALSE;
	timerCollision.IN := TRUE;
	timerCollision.PT := T#2S;
ELSIF collisionSolutionWorking THEN
	CollisionsSolution_new();
END_IF

//Camera damit immer Daten da
IF camera.cameraData.robotPositionArray[Var_HAWIno.Robot_Number].x <> 0 AND camera.cameraData.robotPositionArray[Var_HAWIno.Robot_Number].y <> 0 THEN
	actualCamX := camera.cameraData.robotPositionArray[Var_HAWIno.Robot_Number].x;
	actualCamY := camera.cameraData.robotPositionArray[Var_HAWIno.Robot_Number].y;
END_IF

////////////////////////////////////////////////////////StateMaschine/////////////////////////////////////////////////

//Init
IF sStart AND NOT s0 THEN
	lastRelevantStateForCollision := 's0';
	sStart := 0; s0 := 1;
	//	RückmeldungGW1 Verfügbar
	FeedbackToGW1 := 'Verfuegbar';
	resetVarMQTT := FALSE;
	TrajectoryController.xBoReset := FALSE;
END_IF

//////////////////////////////////////////////////////////////////////////////////////////////////////////////
//////////////////////////////////FAHRAUFTRAG/////////////////////////////////////////////////////////////////
//////////////////////////////////////////////////////////////////////////////////////////////////////////////

//	Warten auf Auftrag
IF s0 AND NOT s1a AND Auftrag.Art = 'Fahrauftrag' THEN
	s0 := 0; s1a := 1;
	lastRelevantStateForCollision := 's1a';
	FeedbackToGW1 := 'Auftrag angenommen';
	//Auftrag auswerten
	readAssigment(assigment:= Auftrag);
	EndNode := readAssigment.endNodePickup;															
	xEndvalue := readAssigment.pickupLocation.x;
	yEndvalue := readAssigment.pickupLocation.y;
	xRobotStartposition := camera.cameraData.robotPositionArray[Var_HAWIno.Robot_Number].x;
	yRobotStartposition := camera.cameraData.robotPositionArray[Var_HAWIno.Robot_Number].y;	
END_IF

//Bahnplanung
IF s1a AND NOT s1b AND xRobotStartposition <> 0 AND yRobotStartposition <> 0 THEN
	AStar(xRobotActual := xRobotStartposition, yRobotActual := yRobotStartposition, xEnd := xEndvalue, yEnd := yEndvalue, endNode := EndNode, blockedNodes := removeNodeCollision);
	finished_ASearch := AStar.finishedASearch;
	IF finished_ASearch THEN
		xPointList := AStar.xCoordinates;
		yPointList := AStar.yCoordinates;
		s1a := 0; s1b := 1;
	END_IF
ELSIF s1a AND NOT s1b THEN
	xRobotStartposition := actualCamX;
	yRobotStartposition := actualCamY;
END_IF

IF s1b AND NOT s2 AND finished_ASearch THEN
	ZEROS_RobotPoseSimple(wayPointList);
	ZEROS_INT(removeNodeCollision);
	finished_ASearch := FALSE;
	FOR i := 0 TO 100 BY 1 DO
 		wayPointList[i] := ToRobotPoseSimple(x:= xPointList[i], y:= yPointList[i], theta:= -1);
		IF xPointList[i] = 0 THEN
			zeile := i;
			EXIT;
		END_IF
	END_FOR
	wayPointList[zeile] := readAssigment.pickupLocation;
	wayPointList[zeile+1] := ToRobotPoseSimple(x := -1, y := -1, theta := -1);
	TrajectoryController.setWaypointList(waypointList);
	trajectoryController.newWaypointListAvailable := TRUE;
	s1b := 0; s2 := 1;
END_IF

///////////////////////////////////////////////FahrtZumAbholort///////////////////////////////////////////////////

// 	RückmeldungGW3 Wegpunkte erhalten abwarten
IF s2 AND NOT s3 AND trajectoryController.yControllerState = ControllerState.setTrajectory THEN
	s2 := 0; s3 := 1;
	trajectoryController.newWaypointListAvailable := FALSE;
END_IF

// 	RückmeldungGW3 ready abwarten
IF s3 AND NOT s4 AND trajectoryController.yControllerState = ControllerState.ready THEN
	s3 := 0; s4 := 1;
	trajectoryController.xBoEnable := TRUE;
END_IF
	
//	RückmeldungGW3 Fahrt abwarten
IF s4 AND NOT s5 AND trajectoryController.yControllerState = ControllerState.driving THEN
	s4 := 0; s5 := 1;
	FeedbackToGW1 := 'Auf Anfahrt';
END_IF

//	RückmeldungGW3 am Ziel abwarten
IF s5 AND NOT s6a AND trajectoryController.yBoArrivedAtDestination THEN
	lastRelevantStateForCollision := 's6a';
	trajectoryController.xBoEnable := FALSE;
	//	Greifersteuerung
	IF NOT Gripper.partGripped THEN
		closeGripperCommand := TRUE;
		s5 := 0; s6a := 1;
	END_IF
END_IF
												
IF s6a AND NOT s6b AND NOT Gripper.partGripped THEN
	s6a := 0; s6b := 1;	
	lastRelevantStateForCollision := 's6b';
	FeedbackToGW1 := 'Teil aufgenommen';
	//	Fahrauftrag zu Lesekopf
	ZEROS_RobotPoseSimple(wayPointList);
	wayPointList := readAssigment.pointsFromSlotToReader;
	TrajectoryController.setWaypointList(wayPointList);
	trajectoryController.newWaypointListAvailable := TRUE;
END_IF


/////////////////////////////////////////////////////FahrtZumLesekopf/////////////////////////////////////////////////////////

// 	RückmeldungGW3 Wegpunkte erhalten abwarten
IF s6b AND NOT s7 AND trajectoryController.yControllerState = ControllerState.setTrajectory AND gripper.state = CoreGripperControlState.Open THEN
	s6b := 0; s7 := 1;
	trajectoryController.newWaypointListAvailable := FALSE;
END_IF

// 	RückmeldungGW3 ready abwarten
IF s7 AND NOT s8 AND trajectoryController.yControllerState = ControllerState.ready THEN
	s7 := 0; s8 := 1;
	trajectoryController.xBoEnable := TRUE;
END_IF
	
//	RückmeldungGW3 Fahrt abwarten
IF s8 AND NOT s9 AND trajectoryController.yControllerState = ControllerState.driving THEN
	s8 := 0; s9 := 1;
	resetVarMQTT := TRUE;
END_IF

//	RückmeldungGW3 am Ziel abwarten
IF s9 AND NOT s10 AND trajectoryController.yBoArrivedAtDestination THEN
	s9 := 0; s10 := 1;
	lastRelevantStateForCollision := 's10';
	trajectoryController.xBoEnable := FALSE;
	resetVarMQTT := FALSE;
	FeedbackToGW1 := 'Abmeldung';
END_IF

IF s10 AND NOT s11a AND StatusFromGW1 = 'WerkstueckAusgelesen' THEN
	s10 := 0; s11a := 1;
	lastRelevantStateForCollision := 's11a';
	//Auftrag auswerten
	EndNode   := readAssigment.endNodeStorage;																	
	xEndvalue := readAssigment.storageLocation.x;
	yEndvalue := readAssigment.storageLocation.y;
	yRobotStartposition := camera.cameraData.robotPositionArray[Var_HAWIno.Robot_Number].y;	
	xRobotStartposition := camera.cameraData.robotPositionArray[Var_HAWIno.Robot_Number].x;
END_IF

//Bahnplanung
IF s11a AND NOT s11b AND xRobotStartposition <> 0 AND yRobotStartposition <> 0 THEN
	AStar(xRobotActual := xRobotStartposition, yRobotActual := yRobotStartposition, xEnd := xEndvalue, yEnd := yEndvalue, endNode := EndNode, blockedNodes := removeNodeCollision);
	finished_ASearch := AStar.finishedASearch;
	IF finished_ASearch THEN
		xPointList := AStar.xCoordinates;
		yPointList := AStar.yCoordinates;
		s11a := 0; s11b := 1;
	END_IF
ELSIF s11a AND NOT s11b THEN
	xRobotStartposition := actualCamX;
	yRobotStartposition := actualCamY;
END_IF

IF s11b AND NOT s12 AND finished_ASearch THEN
	ZEROS_RobotPoseSimple(wayPointList);
	ZEROS_INT(removeNodeCollision);
	finished_ASearch := FALSE;
	FOR i := 0 TO 100 BY 1 DO
 		wayPointList[i] := ToRobotPoseSimple(x:= xPointList[i], y:= yPointList[i], theta:= -1);
		IF xPointList[i] = 0 THEN
			zeile := i;
			EXIT;
		END_IF
	END_FOR
	wayPointList[zeile] := readAssigment.readerCheckIn;
	wayPointList[zeile+1] := ToRobotPoseSimple(x := -1, y := -1, theta := -1);
	TrajectoryController.setWaypointList(waypointList);
	trajectoryController.newWaypointListAvailable := TRUE;
	s11b := 0; s12 := 1;
END_IF

/////////////////////////////////////////////////FahrtZurAblageStation///////////////////////////////////////////////////

// 	RückmeldungGW3 Wegpunkte erhalten abwarten
IF s12 AND NOT s13 AND trajectoryController.yControllerState = ControllerState.setTrajectory THEN
	s12 := 0; s13 := 1;
	trajectoryController.newWaypointListAvailable := FALSE;
END_IF

// 	RückmeldungGW3 ready abwarten
IF s13 AND NOT s14 AND trajectoryController.yControllerState = ControllerState.ready THEN
	s13 := 0; s14 := 1;
	trajectoryController.xBoEnable := TRUE;
END_IF
	
//	RückmeldungGW3 Fahrt abwarten
IF s14 AND NOT s15 AND trajectoryController.yControllerState = ControllerState.driving THEN
	s14 := 0; s15 := 1;
	resetVarMQTT := TRUE;
	FeedbackToGW1 := 'Auf Transport';
END_IF

//	RückmeldungGW3 am Ziel abwarten
IF s15 AND NOT s16 AND trajectoryController.yBoArrivedAtDestination THEN
	s15 := 0; s16 := 1;
	lastRelevantStateForCollision := 's16';	
	trajectoryController.xBoEnable := FALSE;
	resetVarMQTT := FALSE;
	FeedbackToGW1 := 'Anmeldung';
END_IF

//	Warten auf Werkstück ausgelesen
IF s16 AND NOT s17 AND StatusFromGW1 = 'WerkstueckAusgelesen' THEN
	s16 := 0; s17 := 1;
	lastRelevantStateForCollision := 's17';
	//	Fahrauftrag zur Ablage
	ZEROS_RobotPoseSimple(wayPointList);
	wayPointList := readAssigment.pointsFromReaderToSlot;
	TrajectoryController.setWaypointList(wayPointList);
	trajectoryController.newWaypointListAvailable := TRUE;
END_IF

//////////////////////////////////////////////////FahrtZurAblage///////////////////////////////////////////////////////

// 	RückmeldungGW3 Wegpunkte erhalten abwarten
IF s17 AND NOT s18 AND trajectoryController.yControllerState = ControllerState.setTrajectory THEN
	s17 := 0; s18 := 1;
	trajectoryController.newWaypointListAvailable := FALSE;
END_IF

// 	RückmeldungGW3 ready abwarten
IF s18 AND NOT s19 AND trajectoryController.yControllerState = ControllerState.ready THEN
	s18 := 0; s19 := 1;
	trajectoryController.xBoEnable := TRUE;
END_IF
	
//	RückmeldungGW3 Fahrt abwarten
IF s19 AND NOT s20 AND trajectoryController.yControllerState = ControllerState.driving THEN
	s19 := 0; s20 := 1;
	resetVarMQTT := TRUE;
END_IF

//	RückmeldungGW3 am Ziel abwarten
IF s20 AND NOT s21a AND trajectoryController.yBoArrivedAtDestination THEN
	s20 := 0; s21a := 1;
	resetVarMQTT := FALSE;
	lastRelevantStateForCollision := 's21a';
	trajectoryController.xBoEnable := FALSE;
	//	Greifersteuerung
	closeGripperCommand := FALSE;
	FeedbackToGW1 := 'Teil abgelegt';
	//	Fahrauftrag zum Parkplatz
	EndNode := readAssigment.endNodeParking[Var_HAWIno.Robot_Number];															
	xEndvalue := readAssigment.parkingSlots[Var_HAWIno.Robot_Number].x;
	yEndvalue := readAssigment.parkingSlots[Var_HAWIno.Robot_Number].y;
	xRobotStartposition := camera.cameraData.robotPositionArray[Var_HAWIno.Robot_Number].x;
	yRobotStartposition := camera.cameraData.robotPositionArray[Var_HAWIno.Robot_Number].y;	
END_IF

				
//////////////////////////////////////////////////////////////////////////////////////////////////////////////
///////////////////////////////////////LADEAUFTRAG////////////////////////////////////////////////////////////
//////////////////////////////////////////////////////////////////////////////////////////////////////////////

IF s0 AND NOT s26a AND Auftrag.Art = 'Ladeauftrag' THEN
	s0 := 0; s26a := 1;
	lastRelevantStateForCollision := 's26a';
	FeedbackToGW1 := 'Auftrag angenommen';
	//Auftrag auswerten
	readAssigment(assigment:= Auftrag);
	EndNode := readAssigment.endNodeCharging;
	xEndvalue := readAssigment.chargingLocation.x;
	yEndvalue := readAssigment.chargingLocation.y;
	xRobotStartposition := camera.cameraData.robotPositionArray[Var_HAWIno.Robot_Number].x;
	yRobotStartposition := camera.cameraData.robotPositionArray[Var_HAWIno.Robot_Number].y;	
END_IF

//Bahnplanung
IF s26a AND NOT s26b AND xRobotStartposition <> 0 AND yRobotStartposition <> 0 THEN
	AStar(xRobotActual := xRobotStartposition, yRobotActual := yRobotStartposition, xEnd := xEndvalue, yEnd := yEndvalue, endNode := EndNode, blockedNodes := removeNodeCollision);
	finished_ASearch := AStar.finishedASearch;
	IF finished_ASearch THEN
		xPointList := AStar.xCoordinates;
		yPointList := AStar.yCoordinates;
		s26a := 0; s26b := 1;
	END_IF
ELSIF s26a AND NOT s26b THEN
	xRobotStartposition := actualCamX;
	yRobotStartposition := actualCamY;
END_IF

IF s26b AND NOT s27 AND finished_ASearch THEN
	ZEROS_RobotPoseSimple(wayPointList);
	ZEROS_INT(removeNodeCollision);
	finished_ASearch := FALSE;
	FOR i := 0 TO 100 BY 1 DO
 		wayPointList[i] := ToRobotPoseSimple(x:= xPointList[i], y:= yPointList[i], theta:= -1);
		IF xPointList[i] = 0 THEN
			zeile := i;
			EXIT;
		END_IF
	END_FOR
	wayPointList[zeile] := readAssigment.chargingLocation;
	wayPointList[zeile+1] := ToRobotPoseSimple(x := -1, y := -1, theta := -1);
	TrajectoryController.setWaypointList(waypointList);
	trajectoryController.newWaypointListAvailable := TRUE;
	resetVarMQTT := TRUE;														
	s26b := 0; s27 := 1;
END_IF

///////////////////////////////////////////////FahrtZurStation///////////////////////////////////////////////////

// 	RückmeldungGW3 Wegpunkte erhalten abwarten
IF s27 AND NOT s28 AND trajectoryController.yControllerState = ControllerState.setTrajectory THEN
	s27 := 0; s28 := 1;
	trajectoryController.newWaypointListAvailable := FALSE;
END_IF

// 	RückmeldungGW3 ready abwarten
IF s28 AND NOT s29 AND trajectoryController.yControllerState = ControllerState.ready THEN
	s28 := 0; s29 := 1;
	trajectoryController.xBoEnable := TRUE;
END_IF
	
//	RückmeldungGW3 Fahrt abwarten
IF s29 AND NOT s30 AND trajectoryController.yControllerState = ControllerState.driving THEN
	s29 := 0; s30 := 1;
	FeedbackToGW1 := 'Auf Anfahrt';
END_IF

//	RückmeldungGW3 am Ziel abwarten
IF s30 AND NOT s31 AND trajectoryController.yBoArrivedAtDestination THEN
	s30 := 0; s31 := 1;
	lastRelevantStateForCollision := 's31';
	trajectoryController.xBoEnable := FALSE;
	resetVarMQTT := FALSE;					
	FeedbackToGW1 := 'An Ladestation';
END_IF

IF s31 AND NOT s32 AND StatusFromGW1 = 'FertigGeladen' THEN
	s31 := 0; s32 := 1;
	lastRelevantStateForCollision := 's32';
	//	Fahrauftrag von Ladestation weg 
	ZEROS_RobotPoseSimple(wayPointList);
	ZEROS_INT(removeNodeCollision);
	wayPointList[0] := readAssigment.lastNodeCharging;
	wayPointList[1] := ToRobotPoseSimple(x := -1, y := -1, theta := -1); 
	TrajectoryController.setWaypointList(waypointList);
	trajectoryController.newWaypointListAvailable := TRUE;
	resetVarMQTT := TRUE;									
END_IF
	
// 	RückmeldungGW3 Wegpunkte erhalten abwarten
IF s32 AND NOT s33 AND trajectoryController.yControllerState = ControllerState.setTrajectory THEN
	s32 := 0; s33 := 1;
	trajectoryController.newWaypointListAvailable := FALSE;
END_IF

// 	RückmeldungGW3 ready abwarten
IF s33 AND NOT s34 AND trajectoryController.yControllerState = ControllerState.ready THEN
	s33 := 0; s34 := 1;
	trajectoryController.xBoEnable := TRUE;
END_IF
	
//	RückmeldungGW3 Fahrt abwarten
IF s34 AND NOT s35 AND trajectoryController.yControllerState = ControllerState.driving THEN
	s34 := 0; s35 := 1;
END_IF

//	RückmeldungGW3 am Ziel abwarten
IF s35 AND NOT s21a AND trajectoryController.yBoArrivedAtDestination THEN
	s35 := 0; s21a := 1;
	lastRelevantStateForCollision := 's21a';
	trajectoryController.xBoEnable := FALSE;
	resetVarMQTT := FALSE;				
	FeedbackToGW1 := 'Verfuegbar';
	EndNode := readAssigment.endNodeParking[Var_HAWIno.Robot_Number];															
	xEndvalue := readAssigment.parkingSlots[Var_HAWIno.Robot_Number].x;
	yEndvalue := readAssigment.parkingSlots[Var_HAWIno.Robot_Number].y;
	xRobotStartposition := camera.cameraData.robotPositionArray[Var_HAWIno.Robot_Number].x;
	yRobotStartposition := camera.cameraData.robotPositionArray[Var_HAWIno.Robot_Number].y;	
END_IF


//////////////////////////////////////////////////////////////////////////////////////////////////////////////
///////////////////////////////////////Parkplatzanfahrt///////////////////////////////////////////////////////
//////////////////////////////////////////////////////////////////////////////////////////////////////////////

//Bahnplanung
IF s21a AND NOT s21b AND xRobotStartposition <> 0 AND yRobotStartposition <> 0 AND gripper.state = CoreGripperControlState.Closed THEN
	AStar(xRobotActual := xRobotStartposition, yRobotActual := yRobotStartposition, xEnd := xEndvalue, yEnd := yEndvalue, endNode := EndNode, blockedNodes := removeNodeCollision);
	finished_ASearch := AStar.finishedASearch;
	IF finished_ASearch THEN
		xPointList := AStar.xCoordinates;
		yPointList := AStar.yCoordinates;
		s21a := 0; s21b := 1;
	END_IF
ELSIF s21a AND NOT s21b THEN
	xRobotStartposition := actualCamX;
	yRobotStartposition := actualCamY;
END_IF

IF s21b AND NOT s22 AND finished_ASearch THEN
	ZEROS_RobotPoseSimple(wayPointList);
	ZEROS_INT(removeNodeCollision);
	finished_ASearch := FALSE;
	FOR i := 0 TO 100 BY 1 DO
 		wayPointList[i] := ToRobotPoseSimple(x:= xPointList[i], y:= yPointList[i], theta:= -1);
		IF xPointList[i] = 0 THEN
			zeile := i;
			EXIT;
		END_IF
	END_FOR
	wayPointList[zeile] := readAssigment.parkingSlots[Var_HAWIno.Robot_Number];
	wayPointList[zeile+1] := ToRobotPoseSimple(x := -1, y := -1, theta := -1);
	TrajectoryController.setWaypointList(waypointList);
	trajectoryController.newWaypointListAvailable := TRUE;
	s21b := 0; s22 := 1;
END_IF


///////////////////////////////////////////////////FahrtZumParkplatz////////////////////////////////////////////////////////
 
// 	RückmeldungGW3 Wegpunkte erhalten abwarten
IF s22 AND NOT s23 AND trajectoryController.yControllerState = ControllerState.setTrajectory THEN
	s22 := 0; s23 := 1;
	trajectoryController.newWaypointListAvailable := FALSE;
END_IF

// 	RückmeldungGW3 ready abwarten
IF s23 AND NOT s24 AND trajectoryController.yControllerState = ControllerState.ready THEN
	s23 := 0; s24 := 1;
	trajectoryController.xBoEnable := TRUE;
END_IF
	
//	RückmeldungGW3 Fahrt abwarten
IF s24 AND NOT s25 AND trajectoryController.yControllerState = ControllerState.driving THEN
	s24 := 0; s25 := 1;
	//kann schon nächsten Auftrag annehmen
	FeedbackToGW1 := 'Verfuegbar';
END_IF

IF s25 AND NOT s25b AND trajectoryController.yControllerState = ControllerState.driving AND Auftrag.Art = 'Fahrauftrag' THEN
	lastRelevantStateForCollision := 's0';
	trajectoryController.xBoEnable := FALSE;
	s25 := 0; s25b := 1;
END_IF

IF s25b AND NOT s0 AND trajectoryController.yControllerState = ControllerState.ready THEN
	s25b := 0; s0 := 1;
END_IF

//	RückmeldungGW3 am Ziel abwarten
IF s25 AND NOT s0 AND trajectoryController.yBoArrivedAtDestination THEN
	s25 := 0; s0 := 1;
	lastRelevantStateForCollision := 's0';
	trajectoryController.xBoEnable := FALSE;
	FeedbackToGW1 := 'Verfuegbar';
END_IF

////////////////////////////////////////////////////////RESET und ERROR/////////////////////////////////////////////////////

//nur Reset wenn nicht an der Ladestation
IF reset AND NOT s31 THEN 
	TrajectoryController.xBoEnable := FALSE;
	doReset();
	resetTimer.PT := T#1S;
	resetTimer.IN := TRUE;
END_IF

IF Auftrag.Art = '' AND (trajectoryController.yControllerState = ControllerState.idle OR trajectoryController.yControllerState = ControllerState.ready) AND resetTimer.Q THEN
	//reset zurücksetzen, wenn geresettet
	resetTimer.IN := FALSE;
	reset := FALSE;
	readAssigment(assigment := Auftrag);
	EndNode := readAssigment.endNodeParking[Var_HAWIno.Robot_Number];									
	xEndvalue := readAssigment.parkingSlots[Var_HAWIno.Robot_Number].x;
	yEndvalue := readAssigment.parkingSlots[Var_HAWIno.Robot_Number].y;
	xRobotStartposition := camera.cameraData.robotPositionArray[Var_HAWIno.Robot_Number].x;
	yRobotStartposition := camera.cameraData.robotPositionArray[Var_HAWIno.Robot_Number].y;	
	s21a := TRUE;
	lastRelevantStateForCollision := 's21a';
	resetVarMQTT := FALSE;
	TrajectoryController.xBoReset := FALSE;
END_IF

IF AStar.AStarFailed THEN
	failedCounter := failedCounter + 1;
ELSE
	failedCounter := 1;
END_IF

METHOD CameraDataSaved : BOOL
VAR_INPUT
END_VAR

VAR
	n: INT;
END_VAR
//Sicherstellen, dass immer Kameradaten ungleich Null da sind
FOR n := 1 TO 4 BY 1 DO
	IF camera.cameraData.robotPositionArray[n].x <> 0 AND camera.cameraData.robotPositionArray[n].y <> 0 THEN
		cameraX[n] := camera.cameraData.robotPositionArray[n].x;
		cameraY[n] := camera.cameraData.robotPositionArray[n].y;
	END_IF
END_FOR
END_METHOD

METHOD CollisionsSolution_new : BOOL
VAR_INPUT
END_VAR
VAR
	n, higherXRobo, lowerXRobo : INT;
END_VAR
otherRoboInfo();
collisionSolutionWorking := TRUE;

/////////////////////////////////////////////////////////////////NORMAL////////////////////////////////////////////////////////////////////////

IF sk0 AND NOT sk1 AND NOT otherRoboAtStation AND NOT thisRoboAtStation AND NOT otherRoboAtStop AND timerCollision.Q THEN
	todo := 'Warten';
	//darf ich fahren? nur wenn kleinere Roboternummer
	FOR n := 0 TO 4 BY 1 DO
		IF otherRobo[n] > Var_HAWIno.Robot_Number THEN
			todo := 'Fahren';
		END_IF
	END_FOR
	sk0 := 0; sk1 := 1;
	timerCollision.IN := FALSE;
END_IF

IF sk1 AND NOT sk2 AND todo = 'Fahren' THEN
	findNodesToRemove(collisionRobo := otherRobo);
	
	//in richtigen State zurück zum neuplanen und weiterfahren
	xRobotStartposition := camera.cameraData.robotPositionArray[Var_HAWIno.Robot_Number].x;
	yRobotStartposition := camera.cameraData.robotPositionArray[Var_HAWIno.Robot_Number].y;	
	continueAfterCollision();
	todo := '';
	sk1 := 0; sk2 := 1;
END_IF

IF sk1 AND NOT sk3 AND todo = 'Warten' THEN
	sk1 := 0; sk3 := 1;
END_IF

IF sk3 AND NOT sk4 AND collisionFree THEN
	xRobotStartposition := camera.cameraData.robotPositionArray[Var_HAWIno.Robot_Number].x;
	yRobotStartposition := camera.cameraData.robotPositionArray[Var_HAWIno.Robot_Number].y;
	continueAfterCollision();
	todo := '';
	sk3 := 0; sk4 := 1;
END_IF

IF sk2 OR sk4 THEN
	sk2 := 0; sk4 := 0; 
	resetCollision();
END_IF


/////////////////////////////////////////////////////////////ATSTOP////////////////////////////////////////////////////////////////////////////

IF sk0 AND NOT sk10 AND otherRoboAtStop AND timerCollision.Q THEN
	findNodesToRemove(collisionRobo := otherRobo);
	
	xRobotStartposition := camera.cameraData.robotPositionArray[Var_HAWIno.Robot_Number].x;
	yRobotStartposition := camera.cameraData.robotPositionArray[Var_HAWIno.Robot_Number].y;
	continueAfterCollision();
	timerCollision.IN := FALSE;
	sk0 := 0; sk10 := 1;
END_IF

IF sk10 THEN
	sk10 := 0;
	resetCollision();
END_IF


//////////////////////////////////////////////////////////////ATSTATION///////////////////////////////////////////////////////////////////////////

IF sk0 AND NOT sk20 AND (otherRoboAtStation OR thisRoboAtStation) AND timerCollision.Q THEN
	sk0 := 0; sk20 := 1;
	timerCollision.IN := FALSE;
END_IF

//nur anderer Robo an Station
IF sk20 AND NOT sk21 AND otherRoboAtStation AND NOT thisRoboAtStation THEN
	drivingBack();
	IF resetGoBack THEN
		sk20 := 0; sk21 := 1;
	END_IF
END_IF

IF sk21 AND NOT sk22 AND NOT otherRoboAtStation THEN
	xRobotStartposition := camera.cameraData.robotPositionArray[Var_HAWIno.Robot_Number].x;
	yRobotStartposition := camera.cameraData.robotPositionArray[Var_HAWIno.Robot_Number].y;
	continueAfterCollision();
	sk21 := 0; sk22 := 1;
END_IF

//nur dieser Robo an Station
IF sk20 AND NOT sk23 AND NOT otherRoboAtStation AND thisRoboAtStation THEN
	findNodesToRemove(collisionRobo := otherRobo);
	
	//in richtigen State zurück zum neuplanen und weiterfahren
	xRobotStartposition := camera.cameraData.robotPositionArray[Var_HAWIno.Robot_Number].x;
	yRobotStartposition := camera.cameraData.robotPositionArray[Var_HAWIno.Robot_Number].y;	
	continueAfterCollision();
	sk20 := 0; sk23 := 1;
END_IF

//beide an Station
IF sk20 AND NOT sk24 AND otherRoboAtStation AND thisRoboAtStation THEN
	sk20 := 0; sk24 := 1;
	//checken, ob an gleicher Station
	higherXRobo := SEL((camera.cameraData.robotPositionArray[Var_HAWIno.Robot_Number].x > camera.cameraData.robotPositionArray[otherRobo[0]].x), otherRobo[0], Var_HAWIno.Robot_Number);
	lowerXRobo := SEL((camera.cameraData.robotPositionArray[Var_HAWIno.Robot_Number].x < camera.cameraData.robotPositionArray[otherRobo[0]].x), otherRobo[0], Var_HAWIno.Robot_Number);
	IF camera.cameraData.robotPositionArray[higherXRobo].theta > 3 and camera.cameraData.robotPositionArray[higherXRobo].theta < -3 AND camera.cameraData.robotPositionArray[lowerXRobo].theta > -0.1 AND camera.cameraData.robotPositionArray[lowerXRobo].theta < 0.1 THEN
		sameStation := TRUE;
	ELSE
		sameStation := FALSE;
	END_IF  
END_IF

//an gleicher Station
IF sk24 AND NOT sk25 AND sameStation THEN
	xRobotStartposition := camera.cameraData.robotPositionArray[Var_HAWIno.Robot_Number].x;
	yRobotStartposition := camera.cameraData.robotPositionArray[Var_HAWIno.Robot_Number].y;	
	continueAfterCollision();
	sk24 := 0; sk25 := 1;
END_IF

//gleicher Bereich nicht gleiche Station
IF sk24 AND NOT sk26 AND NOT sameStation THEN
	sk24 := 0; sk26 := 1;
END_IF

//dieser Robo auf Transport an Station
IF sk26 AND NOT sk27 AND drivingAtStation THEN
	xRobotStartposition := camera.cameraData.robotPositionArray[Var_HAWIno.Robot_Number].x;
	yRobotStartposition := camera.cameraData.robotPositionArray[Var_HAWIno.Robot_Number].y;	
	continueAfterCollision();
	sk26 := 0; sk27 := 1;
END_IF

//dieser nicht aber anderer auf Transport an Station
IF sk26 AND NOT sk28 AND NOT drivingAtStation AND goBack THEN
	drivingBack();
	IF resetGoBack THEN
		sk26 := 0; sk28 := 1;
	END_IF
END_IF

IF sk28 AND NOT sk29 AND NOT otherRoboAtStation THEN
	xRobotStartposition := camera.cameraData.robotPositionArray[Var_HAWIno.Robot_Number].x;
	yRobotStartposition := camera.cameraData.robotPositionArray[Var_HAWIno.Robot_Number].y;	
	continueAfterCollision();
	sk28 := 0; sk29 := 1;
END_IF

//beide im Stationsbereich und keiner auf Transport an Station - was wenn die hier gegenüber?
IF sk26 AND NOT sk30 AND NOT drivingAtStation AND NOT goBack THEN
	todo := 'Warten';		
	IF SQRT(EXPT(camera.cameraData.robotPositionArray[Var_HAWIno.Robot_Number].x - AStar.xEnd,2) + EXPT(camera.cameraData.robotPositionArray[Var_HAWIno.Robot_Number].x - 2800,2)) < SQRT(EXPT(camera.cameraData.robotPositionArray[otherRobo[0]].x - AStar.xEnd,2) + EXPT(camera.cameraData.robotPositionArray[otherRobo[0]].x - 2800,2)) THEN
		//dieser Robo dichter dran
		todo := 'Fahren';
	END_IF
	sk26 := 0; sk30 := 1;
END_IF

IF sk30 AND NOT sk31 AND todo = 'Fahren' THEN
	xRobotStartposition := camera.cameraData.robotPositionArray[Var_HAWIno.Robot_Number].x;
	yRobotStartposition := camera.cameraData.robotPositionArray[Var_HAWIno.Robot_Number].y;	
	continueAfterCollision();
	sk30 := 0; sk31 := 1;
END_IF

IF sk30 AND NOT sk32 AND todo = 'Warten' THEN
	drivingBack();
	IF resetGoBack THEN
		sk30 := 0; sk32 := 1;
	END_IF
END_IF

IF sk32 AND NOT sk33 AND NOT otherRoboAtStation THEN
	xRobotStartposition := camera.cameraData.robotPositionArray[Var_HAWIno.Robot_Number].x;
	yRobotStartposition := camera.cameraData.robotPositionArray[Var_HAWIno.Robot_Number].y;	
	continueAfterCollision();
	sk30 := 0; sk31 := 1;
END_IF

IF resetGoBack AND NOT goBack THEN
	resetGoBack := FALSE;
END_IF

/////////////////////////////////////////Am Ende der Kollisionsauflösung//////////////////////////////////////////////
IF sk22 OR sk23 OR sk25 OR sk27 OR sk29 OR sk31 OR sk33 THEN
	sk22 := 0; sk23 := 0; sk25 := 0; sk27 := 0; sk29 := 0; sk31 := 0; sk33 := 0;
	resetCollision();
END_IF
END_METHOD

METHOD continueAfterCollision : BOOL
VAR_INPUT
END_VAR
VAR
	diffToList : ARRAY[0..100] OF LREAL;						//Differenz Kamera zu Wegpunktlisten
	sortedDiff : ARRAY[0..100,1..2] OF LREAL;					//sortierte Differenzliste
	nextIndex, j, n, l, i : INT;									
	nullSortedDiff : ARRAY[0..100,1..2] OF LREAL := [202(0)];	//Nullarray zum Zurücksetzen
END_VAR

//nächsten abzuarbeitenden State setzen
IF lastRelevantStateForCollision = 's0' THEN
	s0 := 1;
ELSIF lastRelevantStateForCollision = 's1a' THEN
	s1a := 1;
ELSIF lastRelevantStateForCollision = 's6a' THEN
	s6a := 1;
ELSIF lastRelevantStateForCollision = 's6b' THEN
	s6b := 1;

	//Arrays resetten
	ZEROS(diffToList);
	sortedDiff := nullSortedDiff;
	
	FOR i := 0 TO 10 BY 1 DO
		IF readAssigment.pointsFromSlotToReader[i].x > 0 AND readAssigment.pointsFromSlotToReader[i].y > 0 THEN
			//Abstände Roboter zu Wegpunkten
			diffToList[i] := SQRT(EXPT(camera.cameraData.robotPositionArray[Var_HAWIno.Robot_Number].x - readAssigment.pointsFromSlotToReader[i].x,2) + EXPT(camera.cameraData.robotPositionArray[Var_HAWIno.Robot_Number].y - readAssigment.pointsFromSlotToReader[i].y,2));
			FOR n := 0 TO 10 BY 1 DO
				IF diffToList[i] < sortedDiff[n,2] THEN
					FOR l := 9 TO n BY -1 DO
						sortedDiff[l+1,1] := sortedDiff[l,1];
						sortedDiff[l+1,2] := sortedDiff[l,2];
					END_FOR
					sortedDiff[n,2] := diffToList[i];
					sortedDiff[n,1] := i;
					EXIT;
				ELSIF i = 0 THEN
					sortedDiff[0,2] := diffToList[0];
					sortedDiff[0,1] := 0;
					EXIT;
				END_IF
			END_FOR
		END_IF	
	END_FOR
	
	ZEROS_RobotPoseSimple(wayPointList);
	nextIndex := LREAL_TO_INT(MAX(sortedDiff[0,1],sortedDiff[1,1]));	//Index des nächsten anzufahrenden Wegpunkt
	
	FOR i := 0 TO 100 - nextIndex BY 1 DO 
		wayPointList[i] := readAssigment.pointsFromSlotToReader[nextIndex + i];
	END_FOR 
	TrajectoryController.setWaypointList(wayPointList);
	trajectoryController.newWaypointListAvailable := TRUE;

ELSIF lastRelevantStateForCollision = 's10' THEN
	s10 := 1;
ELSIF lastRelevantStateForCollision = 's11a' THEN
	s11a := 1;
ELSIF lastRelevantStateForCollision = 's16' THEN
	s16 := 1;
ELSIF lastRelevantStateForCollision = 's17' THEN
	s17 := 1;
	
	//Arrays resetten
	ZEROS(diffToList);
	sortedDiff := nullSortedDiff;
	
	FOR i := 0 TO 10 BY 1 DO
		IF readAssigment.pointsFromReaderToSlot[i].x <> 0 AND readAssigment.pointsFromReaderToSlot[i].y <> -1 THEN
			//Abstände Roboter zu Wegpunkten
			diffToList[i] := SQRT(EXPT(camera.cameraData.robotPositionArray[Var_HAWIno.Robot_Number].x - readAssigment.pointsFromReaderToSlot[i].x,2) + EXPT(camera.cameraData.robotPositionArray[Var_HAWIno.Robot_Number].y - readAssigment.pointsFromReaderToSlot[i].y,2));
			FOR n := 0 TO 10 BY 1 DO
				IF diffToList[i] < sortedDiff[n,2] THEN
					FOR l := 9 TO n BY -1 DO
						sortedDiff[l+1,1] := sortedDiff[l,1];
						sortedDiff[l+1,2] := sortedDiff[l,2];
					END_FOR
					sortedDiff[n,2] := diffToList[i];
					sortedDiff[n,1] := i;
					EXIT;
				ELSIF i = 0 THEN
					sortedDiff[0,2] := diffToList[0];
					sortedDiff[0,1] := 0;
					EXIT;
				END_IF
			END_FOR
		END_IF	
	END_FOR
	
	ZEROS_RobotPoseSimple(wayPointList);
	nextIndex := LREAL_TO_INT(MAX(sortedDiff[0,1],sortedDiff[1,1])); 	//Index des nächsten anzufahrenden Wegpunkt
	
	FOR i := 0 TO 100 - nextIndex BY 1 DO 
		wayPointList[i] := readAssigment.pointsFromReaderToSlot[nextIndex + i];
	END_FOR 
	TrajectoryController.setWaypointList(wayPointList);
	trajectoryController.newWaypointListAvailable := TRUE;
	
ELSIF lastRelevantStateForCollision = 's21a' THEN
	s21a := 1;
ELSIF lastRelevantStateForCollision = 's26a' THEN
	s26a := 1;
ELSIF lastRelevantStateForCollision = 's31' THEN
	s31 := 1;
ELSIF lastRelevantStateForCollision = 's32' THEN
	s32 := 1;
END_IF
END_METHOD

METHOD doReset : BOOL
VAR_INPUT
	
END_VAR
resetVarMQTT := TRUE;
TrajectoryController.xBoReset := TRUE;
ZEROS_RobotPoseSimple(wayPointList);
closeGripperCommand := True;
actualCamX := 0;
actualCamY := 0;
trajectoryController.newWaypointListAvailable := FALSE;
trajectoryController.xBoEnable := FALSE;
FeedbackToGW1 := 'Verfuegbar';
closeGripperCommand := FALSE;
ZEROS_INT(removeNodeCollision);
error := FALSE;
failedCounter := 1;

//Statemaschine zurücksetzen
sStart := FALSE;
s0 := FALSE;
s1a := FALSE;
s1b := FALSE;
s2 := FALSE;
s3 := FALSE;
s4 := FALSE;
s5 := FALSE;
s6a := FALSE;
s6b := FALSE;
s7 := FALSE;
s8 := FALSE;
s9 := FALSE;
s10 := FALSE;
s11a := FALSE;
s11b := FALSE;
s12 := FALSE;
s13 := FALSE;
s14 := FALSE;
s15 := FALSE;
s16 := FALSE;
s17 := FALSE;
s18 := FALSE;
s19 := FALSE;
s20 := FALSE;
s21a := FALSE;
s21b := FALSE;
s22 := FALSE;
s23 := FALSE;
s24 := FALSE;
s25 := FALSE;
s26a := FALSE;
s26b := FALSE;
s27 := FALSE;
s28 := FALSE;
s29 := FALSE;
s30 := FALSE;
s31 := FALSE;

resetCollision();
END_METHOD

METHOD drivingBack : BOOL
VAR_INPUT
END_VAR

VAR
	gbWayPointList : ARRAY[0..100] OF RobotPoseSimple;			//goBack Wegpunktliste
	diffToList : ARRAY[0..100] OF LREAL;						//Differenz aktuelle Position und Wegpunktliste
	sortedDiff : ARRAY[0..100,1..2] OF LREAL;					//sortierte Differenzliste
	index, n, l, i : INT;
	camX, camY : LREAL;											//Kameradaten
	alternativeGoAway: BOOL;
	nullSortedDiff : ARRAY[0..100,1..2] OF LREAL := [202(0)];	//zum Zurücksetzen
END_VAR
IF firstTime THEN 
	//Arrays resetten
	ZEROS_RobotPoseSimple(gbWayPointList);
	ZEROS(diffToList);
	sortedDiff := nullSortedDiff;
	alternativeGoAway := FALSE;

	camX := camera.cameraData.robotPositionArray[Var_HAWIno.Robot_Number].x;
	camY := camera.cameraData.robotPositionArray[Var_HAWIno.Robot_Number].y;
	IF camX = 0 AND camY = 0 THEN
		camX := actualCamX;
		camY := actualCamY;
	END_IF
	
	FOR i := 0 TO 100 BY 1 DO
		IF wayPointList[i].x <> 0 AND wayPointList[i].y <> 0 THEN
			//Abstände Roboter zu Wegpunkten
			diffToList[i] := SQRT(EXPT(camX - wayPointList[i].x,2) + EXPT(camY - wayPointList[i].y,2));
			FOR n := 0 TO 100 BY 1 DO
				IF diffToList[i] < sortedDiff[n,2] THEN
					FOR l := 99 TO n BY -1 DO
						sortedDiff[l+1,1] := sortedDiff[l,1];
						sortedDiff[l+1,2] := sortedDiff[l,2];
					END_FOR
					sortedDiff[n,2] := diffToList[i];
					sortedDiff[n,1] := i;
					EXIT;
				ELSIF i = 0 THEN
					sortedDiff[0,2] := diffToList[0];
					sortedDiff[0,1] := 0;
					EXIT;
				ELSIF sortedDiff[n+1,2] = 0 THEN
					sortedDiff[n+1,2] := diffToList[i];
					sortedDiff[n+1,1] := i;
					EXIT;
				END_IF
			END_FOR
		END_IF	
	END_FOR
	
	//Index vom letzten angefahrenen Wegpunkt
	index := LREAL_TO_INT(MIN(sortedDiff[0,1],sortedDiff[1,1]));
	
	IF index > 1 THEN
		gbWaypointList[0] := wayPointList[index];
		gbWaypointList[1] := wayPointList[index-1];
		gbWaypointList[2] := wayPointList[index-2];
		gbWaypointList[3] := ToRobotPoseSimple(x := -1, y := -1, theta := -1);
	ELSE
		alternativeGoAway := TRUE;
	END_IF
	
	TrajectoryController.setWaypointList(gbWaypointList);
	trajectoryController.newWaypointListAvailable := TRUE;
	firstTime := FALSE;
END_IF

IF trajectoryController.yControllerState = ControllerState.setTrajectory THEN
	trajectoryController.newWaypointListAvailable := FALSE;
END_IF

// 	RückmeldungGW3 ready abwarten
IF trajectoryController.yControllerState = ControllerState.ready THEN
	trajectoryController.xBoEnable := TRUE;
END_IF

IF trajectoryController.yBoArrivedAtDestination THEN
	trajectoryController.xBoEnable := FALSE;
	resetGoBack := true;
	firstTime := TRUE;
END_IF
END_METHOD

METHOD errorTest : BOOL
VAR_INPUT
END_VAR
//ERROR: Teil verloren
IF gripper.state = CoreGripperControlState.Open AND Gripper.partGripped THEN
	error := TRUE;
	TrajectoryController.xBoEnable := FALSE;	
	removeAllToken();
	FeedbackToGW1 := 'Error Teil verloren';
	closeGripperCommand := FALSE;
	resetVarMQTT := FALSE;
END_IF
	
//ERROR: Error von GW3
IF trajectoryController.yControllerState = ControllerState.error THEN
	error := TRUE;
	removeAllToken();
	FeedbackToGW1 := 'Error Bumper';
	closeGripperCommand := FALSE;
	resetVarMQTT := FALSE;
END_IF

//wenn AStern auch nach 1000 Zyklen immernoch Failed
IF failedCounter > 1000 THEN
	error := TRUE;
	FeedbackToGW1 := 'Fehler AStar';
	closeGripperCommand := FALSE;
	resetVarMQTT := FALSE;
END_IF
END_METHOD

METHOD findNodesToRemove : BOOL
VAR_INPUT
	collisionRobo : ARRAY[0..4] OF INT;						//an Kollision beteiligte Roboter
END_VAR
VAR
	xMinBox, xMaxBox, yMinBox, yMaxBox, row, col : LREAL;	
	xNode, yNode : ARRAY[1..170] OF LREAL;					//Koordinaten der Knoten
	d, j, w : INT;
END_VAR
w := 1;

FOR d := 0 TO 4 BY 1 DO
	IF collisionRobo[d] <> 0 THEN
		//Umrechnung von Knoten in Koordinaten
		 row := 600;
		 col := 200;
		 
		 FOR i := 1 TO 144 BY 1 DO
			 IF xNode[i] <> 10000 THEN
				xNode[i] := col;
			 END_IF
			 IF yNode[i] <> 10000 THEN
				yNode[i] := row;
			 END_IF
			 col := col + 400;
			 IF i MOD 18 = 0 THEN
				 col := 200;
				 row := row + 400;
			 END_IF
		 END_FOR
		 
		 xNode[145] := 850;
		 xNode[146] := 850;
		 xNode[147] := 850;
		 xNode[148] := 1350;
		 xNode[149] := 1350;
		 xNode[150] := 1350;
		 xNode[151] := 2050;
		 xNode[152] := 2050;
		 xNode[153] := 2050;
		 xNode[154] := 2490;
		 xNode[155] := 2490;
		 xNode[156] := 2490;
		 xNode[157] := 3190;
		 xNode[158] := 3190;
		 xNode[159] := 3190;
		 xNode[160] := 3700;
		 xNode[161] := 3700;
		 xNode[162] := 3700;
		 xNode[163] := 4420;
		 xNode[164] := 4420;
		 xNode[165] := 4420;
		 xNode[166] := 4940;
		 xNode[167] := 4940;
		 xNode[168] := 4940;
		 xNode[169] := 6117;
		 xNode[170] := 6716;
		 
		 yNode[145] := 2735;
		 yNode[146] := 2838;
		 yNode[147] := 2936;
		 yNode[148] := 2736;
		 yNode[149] := 2835;
		 yNode[150] := 2935;
		 yNode[151] := 2731;
		 yNode[152] := 2829;
		 yNode[153] := 2931;
		 yNode[154] := 2732;
		 yNode[155] := 2833;
		 yNode[156] := 2928;
		 yNode[157] := 2732;
		 yNode[158] := 2837;
		 yNode[159] := 2940;
		 yNode[160] := 2732;
		 yNode[161] := 2840;
		 yNode[162] := 2940;
		 yNode[163] := 2732;
		 yNode[164] := 2838;
		 yNode[165] := 2944;
		 yNode[166] := 2746;
		 yNode[167] := 2855;
		 yNode[168] := 2942;
		 yNode[169] := 3450;
		 yNode[170] := 3450;
		 
		
		//im Abstand von 400 all Knoten um Robot löschen
		IF camera.cameraData.robotPositionArray[collisionRobo[d]].x <> 0 AND camera.cameraData.robotPositionArray[collisionRobo[d]].y <> 0 THEN
			xMinBox := camera.cameraData.robotPositionArray[collisionRobo[d]].x - 400;
			xMaxBox := camera.cameraData.robotPositionArray[collisionRobo[d]].x + 400;
			yMinBox := camera.cameraData.robotPositionArray[collisionRobo[d]].y - 400;
			yMaxBox := camera.cameraData.robotPositionArray[collisionRobo[d]].y + 400;
		ELSE 
			xMinBox := cameraX[collisionRobo[d]] - 400;
			xMaxBox := cameraX[collisionRobo[d]] + 400;
			yMinBox := cameraY[collisionRobo[d]] - 400;
			yMaxBox := cameraY[collisionRobo[d]] + 400;
		END_IF
		
		FOR j := 1 TO 170 BY 1 DO
			IF xNode[j] > xMinBox AND xNode[j] < xMaxBox AND yNode[j] > yMinBox AND yNode[j] < yMaxBox THEN
				removeNodeCollision[w] := j;
				w := w + 1;
			END_IF
		END_FOR
	END_IF
END_FOR
END_METHOD

METHOD otherRoboInfo : BOOL
VAR_INPUT
END_VAR
VAR
	nmb, z: INT;
END_VAR
CameraDataSaved();			//Sicherstellen, dass immer Kameradaten und nicht Null

IF newCollision THEN
	removeAllToken();
	i := 0;
	//beteiligte Roboter finden
	FOR nmb := 0 TO 4 BY 1 DO
		IF collision[nmb] AND nmb <> Var_HAWIno.Robot_Number THEN
			otherRobo[i] := nmb;
			i := i + 1;
		END_IF
	END_FOR
END_IF

IF otherRobo[0] > 0 THEN
	IF cameraY[otherRobo[0]] < 650 THEN
		//Anderer Roboter auf Parkplatz
		otherRoboAtStop := TRUE;	
	ELSIF cameraX[otherRobo[0]] > 6100 AND cameraX[otherRobo[0]] < 6800 AND cameraY[otherRobo[0]] > 3400 AND cameraY[otherRobo[0]] < 3600  THEN
		//Anderer Roboter an Ladestation
		otherRoboAtStop := TRUE;
	ELSE
		otherRoboAtStop := FALSE;
	END_IF
	
	IF cameraX[otherRobo[0]] > 0 AND cameraX[otherRobo[0]] < 5200 AND cameraY[otherRobo[0]] > 2340 AND cameraY[otherRobo[0]] < 3345  THEN
		//Anderer Roboter im Bereich der Stationen
		otherRoboAtStation := TRUE;
	ELSE
		otherRoboAtStation := FALSE;
	END_IF
	
	IF cameraX[Var_HAWIno.Robot_Number] > 0 AND cameraX[Var_HAWIno.Robot_Number] < 5200 AND cameraY[Var_HAWIno.Robot_Number] > 2340 AND cameraY[Var_HAWIno.Robot_Number] < 3345  THEN
		//dieser Roboter im Bereich der Stationen
		thisRoboAtStation := TRUE;
	ELSE
		thisRoboAtStation := FALSE;
	END_IF
	
	//Stationsfahrt: anderen Robo wegschicken
	IF lastRelevantStateForCollision = 's6a' OR lastRelevantStateForCollision = 's6b' OR lastRelevantStateForCollision = 's10' OR lastRelevantStateForCollision = 's16' OR lastRelevantStateForCollision = 's17' THEN
		//anderen Wegschicken, weil dieser Roboter auf Transport an Station
		FOR z := 0 TO 4 DO
			IF newCollision AND otherRobo[z] <> 0 THEN
				RoboNmbToGoBack[z] := otherRobo[z];
			ELSIF NOT otherRoboAtStation THEN
				RoboNmbToGoBack[z] := 0;
			END_IF 
			drivingAtStation := TRUE;
		END_FOR
	ELSE
		drivingAtStation := FALSE;
	END_IF
ELSE
	error := TRUE;
	removeAllToken();
END_IF
END_METHOD

METHOD removeAllToken : BOOL
VAR_INPUT
END_VAR
//Statemaschine zurücksetzen
sStart := FALSE;
s0 := FALSE;
s1a := FALSE;
s1b := FALSE;
s2 := FALSE;
s3 := FALSE;
s4 := FALSE;
s5 := FALSE;
s6a := FALSE;
s6b := FALSE;
s7 := FALSE;
s8 := FALSE;
s9 := FALSE;
s10 := FALSE;
s11a := FALSE;
s11b := FALSE;
s12 := FALSE;
s13 := FALSE;
s14 := FALSE;
s15 := FALSE;
s16 := FALSE;
s17 := FALSE;
s18 := FALSE;
s19 := FALSE;
s20 := FALSE;
s21a := FALSE;
s21b := FALSE;
s22 := FALSE;
s23 := FALSE;
s24 := FALSE;
s25 := FALSE;
s26a := FALSE;
s26b := FALSE;
s27 := FALSE;
s28 := FALSE;
s29 := FALSE;
s30 := FALSE;
s31 := FALSE;
END_METHOD

METHOD resetCollision : BOOL
VAR_INPUT
END_VAR
//Kollisionsvariabelen zurücksetzen

collisionSolutionWorking := FALSE; 

Zeros_INT(otherRobo);
otherRoboAtStop := FALSE;
otherRoboAtStation := FALSE;
thisRoboAtStation := FALSE;
RoboNmbToGoBack[0] := 0;
RoboNmbToGoBack[1] := 0;
RoboNmbToGoBack[2] := 0;
RoboNmbToGoBack[3] := 0;
RoboNmbToGoBack[4] := 0;
drivingAtStation := FALSE;
sameStation := FALSE;
todo := '';

sk0 := FALSE;
sk1 := FALSE;
sk2 := FALSE;
sk3 := FALSE;
sk4 := FALSE;
sk10 := FALSE;
sk20 := FALSE;
sk21 := FALSE;
sk22 := FALSE;
sk23 := FALSE;
sk24 := FALSE;
sk25 := FALSE;
sk26 := FALSE;
sk27 := FALSE;
sk28 := FALSE;
sk29 := FALSE;
sk30 := FALSE;
sk31 := FALSE;
sk32 := FALSE;
sk33 := FALSE;
END_METHOD

END_PROGRAM

// ---- POUs/UserPOUs/GW2/AStar.TcPOU
FUNCTION_BLOCK AStar
VAR_INPUT
	xRobotActual, yRobotActual : LREAL;						//aktuelle Roboterposition
	xEnd, yEnd : LREAL;										//Endkoordinaten
	endNode : INT ;											//Endknoten
	blockedNodes : ARRAY[1..11] OF INT;						//geblockte Knoten
END_VAR
VAR_OUTPUT
	finishedASearch, AStarFailed : BOOL := FALSE;			//Erfolg oder Misserfolg von AStern
	xCoordinates, yCoordinates : ARRAY[0..100] OF LREAL;	//Koordinatenliste des Weges
END_VAR
VAR
	//Nullarrays für Zurücksetzen
	nullMatrix_Neighbor : ARRAY[1..8,1..5] OF LREAL := [40(0)];
	nullMatrix_TempArray : ARRAY[1..170,1..7] OF LREAL := [1190(0)];
	nullOpenList : ARRAY[1..170,1..6] OF LREAL := [1020(0)];
	
	numberOfNodes : INT := 144;
	numberOfColumns : INT := 18;
	a, b, c, d, e, i, j, k, m, o, p, q, t, v, w, counter, counter1, number, cnt1, cnt2, cntPark : INT;
	matrix : ARRAY[1..170,1..170] OF LREAL;				//Adjezenzmatrix
	row, col : LREAL;
	xNode, yNode : ARRAY[1..170] OF LREAL;				//Koordinaten der Knoten
	removeNode : ARRAY[0..30] OF INT := [3, 6, 9, 12, 93, 96, 99, 102, 111, 114, 117, 120, 124, 125, 142, 143];	//zu entfernende Knoten
	startNode : INT := 0;
	diff_x, diff_y, diff_total : ARRAY[1..170] OF LREAL;
	min_total : LREAL;
	openList : ARRAY[1..170,1..6] OF LREAL;
	closedList : ARRAY[1..170] OF LREAL;
	h, f, gprev : LREAL;
	g : LREAL := 0;
	parentNode : INT ;
	countNeighbor, indexMin, currentNode : INT;
	neighborList:ARRAY[1..8,1..5] OF LREAL;
	flag : BOOL;
	countOpen : INT := 1;
	tempArray : ARRAY[1..170,1..7] OF LREAL;
	countTemp : INT := 1;
	minf : LREAL;
	wayPointList : ARRAY[1..101] OF INT;
	wayPointList_finished : ARRAY[0..100] OF INT;
	countClosed : INT := 1;
	countPointList : INT := 1;
END_VAR

reset();
openList := nullOpenList;

FOR counter1 := 1 TO 11 DO
	removeNode[15 + counter1] := blockedNodes[counter1];
	
	//Fail, wenn Zielknoten bei entfernten Knoten ist
	IF blockedNodes[counter1] = endNode THEN
		AStarFailed := TRUE;
	END_IF
END_FOR 

///////////////////////////////////////////Erstellen der Adjezenzmatrix//////////////////////////////////////////////////////////////////
FOR i := 0 TO numberOfNodes BY 1 DO
	 IF i-1 > 0 AND i MOD numberOfColumns <> 1 THEN									//linker Nachbar
		 matrix[i-1,i] := 1000;
	 END_IF
	 IF i+1 < numberOfNodes+1 AND i MOD numberOfColumns <> 0 THEN					//rechter Nachbar
		 matrix[i+1,i] := 1000;
	 END_IF
	 IF i+numberOfColumns < numberOfNodes+1 THEN									//oberer Nachbar
		 matrix[i+numberOfColumns,i] := 1000;
	 END_IF
	 IF i-numberOfColumns > 0 THEN													//unterer Nachbar
		 matrix[i-numberOfColumns,i] := 1000;
	 END_IF
	 IF i+numberOfColumns+1 < numberOfNodes+1 AND i MOD numberOfColumns <> 0 THEN	//Nachbar oben rechts
		 matrix[i+numberOfColumns+1,i] := SQRT(2)*1000;
	 END_IF
	 IF i+numberOfColumns-1 < numberOfNodes+1 AND i MOD numberOfColumns <> 1 THEN	//Nachbar oben links
		 matrix[i+numberOfColumns-1,i] := SQRT(2)*1000;
	 END_IF
	 IF i-numberOfColumns+1 > 0 AND i MOD numberOfColumns <> 0 THEN					//Nachbar unten rechts
		 matrix[i-numberOfColumns+1,i] := SQRT(2)*1000;
	 END_IF
	 IF i-numberOfColumns-1 > 0 AND i MOD numberOfColumns <> 1 THEN					//Nachbar unten links
		 matrix[i-numberOfColumns-1,i] := SQRT(2)*1000;
	 END_IF
 END_FOR
 
//Löschen der Knoten über Station und die nahegelegenen diagonalen Verbindungen
 FOR counter := 0 TO 30 BY 1 DO 	
	//Verbindungen zu und um entfernte Knoten entfernen
	IF removeNode[counter] > 0 THEN 
		FOR j := 1 TO 170 BY 1 DO
			matrix[removeNode[counter],j] := 0;
			matrix[j, removeNode[counter]] := 0;
		END_FOR
		
		//diagonale Verbindung oben links
		IF removeNode[counter] - 1 > 0 AND removeNode[counter] + numberOfColumns <= numberOfNodes THEN 
			matrix[removeNode[counter] - 1, removeNode[counter] + numberOfColumns] := 0;	
			matrix[removeNode[counter] + numberOfColumns, removeNode[counter] - 1] := 0;	
		END_IF
		
		//diagonale Verbindung unten links
		IF removeNode[counter] - 1 > 0 AND removeNode[counter] - numberOfColumns > 0 THEN 
			matrix[removeNode[counter] - 1, removeNode[counter] - numberOfColumns] := 0;	
			matrix[removeNode[counter] - numberOfColumns, removeNode[counter] - 1] := 0;	
		END_IF
		
		//diagonale Verbindung oben rechts
		IF removeNode[counter] + 1 <= numberOfNodes AND removeNode[counter] + numberOfColumns <= numberOfNodes THEN 
			matrix[removeNode[counter] + 1, removeNode[counter] + numberOfColumns] := 0;	
			matrix[removeNode[counter] + numberOfColumns, removeNode[counter] + 1] := 0;	
		END_IF
		
		//diagonale Verbindung unten rechts
		IF removeNode[counter] + 1 <= numberOfNodes AND removeNode[counter] - numberOfColumns > 0 THEN
			matrix[removeNode[counter] + 1, removeNode[counter] - numberOfColumns] := 0;	
			matrix[removeNode[counter] - numberOfColumns, removeNode[counter] + 1] := 0;	
		END_IF
		
		//alle entfernten Knoten auf unrealistische Koordinaten setzen, damit sie nicht als Startknoten in Frage kommen, außer die Partplätze
		IF counter > 3 THEN
			xNode[removeNode[counter]] := 10000;
			yNode[removeNode[counter]] := 10000;
		END_IF
	END_IF
 END_FOR
 
 //neue Knoten für Taschenanfahrt
 o := 0;
 FOR number := 1 TO 24 BY 6 DO
	 FOR cnt1 := 0 TO 2 BY 1 DO 
		 matrix[numberOfNodes + number + cnt1, 92 + o] := 1000;
		 matrix[92 + o, numberOfNodes + number + cnt1] := 1000;
		 matrix[numberOfNodes + number + cnt1, 110 + o] := 1000;
		 matrix[110 + o, numberOfNodes + number + cnt1] := 1000;
	END_FOR
	FOR cnt2 := 3 TO 5 BY 1 DO 
		 matrix[numberOfNodes + number + cnt2, 92 + o + 2] := 1000;
		 matrix[92 + o + 2, numberOfNodes + number + cnt2] := 1000;
		 matrix[numberOfNodes + number + cnt2, 110 + o + 2] := 1000;
		 matrix[110 + o + 2, numberOfNodes + number + cnt2] := 1000;
	END_FOR
	o := o + 3;
 END_FOR
 
 matrix[numberOfNodes + number, 106] := 1000;
 matrix[106, numberOfNodes + number] := 1000;
 matrix[numberOfNodes + number + 1, 107] := 1000;
 matrix[107, numberOfNodes + number + 1] := 1000;
 
 //Parkplätze mit nur einer Verbindung
 FOR cntPark := 3 TO 12 BY 3 DO
	 matrix[cntPark, cntPark + 18] := 1000;
	 matrix[cntPark + 18, cntPark] := 1000;
 END_FOR
 
 //Umrechnung von Knoten in Koordinaten
 row := 600;
 col := 200;
 
  FOR i := 1 TO numberOfNodes BY 1 DO
	 IF xNode[i] <> 10000 THEN
	 	xNode[i] := col;
	 END_IF
	 IF yNode[i] <> 10000 THEN
	 	yNode[i] := row;
	 END_IF
	 col := col + 400;
	 IF i MOD numberOfColumns = 0 THEN
		 col := 200;
		 row := row + 400;
	 END_IF
 END_FOR
 
 //nochmal mit pickuplocation und co machen also ohne magic numbers
 xNode[145] := 790;
 xNode[146] := 790;
 xNode[147] := 790;
 xNode[148] := 1410;
 xNode[149] := 1410;
 xNode[150] := 1410;
 xNode[151] := 1990;
 xNode[152] := 1990;
 xNode[153] := 1990;
 xNode[154] := 2550;
 xNode[155] := 2550;
 xNode[156] := 2550;
 xNode[157] := 3130;
 xNode[158] := 3130;
 xNode[159] := 3130;
 xNode[160] := 3760;
 xNode[161] := 3760;
 xNode[162] := 3760;
 xNode[163] := 4360;
 xNode[164] := 4360;
 xNode[165] := 4360;
 xNode[166] := 5000;
 xNode[167] := 5000;
 xNode[168] := 5000;
 xNode[169] := 6117;
 xNode[170] := 6716;
 
 yNode[145] := 2735;
 yNode[146] := 2838;
 yNode[147] := 2936;
 yNode[148] := 2736;
 yNode[149] := 2835;
 yNode[150] := 2935;
 yNode[151] := 2731;
 yNode[152] := 2829;
 yNode[153] := 2931;
 yNode[154] := 2732;
 yNode[155] := 2833;
 yNode[156] := 2928;
 yNode[157] := 2732;
 yNode[158] := 2837;
 yNode[159] := 2940;
 yNode[160] := 2732;
 yNode[161] := 2840;
 yNode[162] := 2940;
 yNode[163] := 2732;
 yNode[164] := 2838;
 yNode[165] := 2944;
 yNode[166] := 2737;
 yNode[167] := 2855;
 yNode[168] := 2942;
 yNode[169] := 3100;
 yNode[170] := 3100;
 
 
 ////////////////////////////////////////////////////Startposition und Endposition bestimmen //////////////////////////////////////////////////////////////////////////
 
 FOR i := 1 TO 170 BY 1 DO
	 diff_x[i] := ABS(xRobotActual - xNode[i]);
	 diff_y[i] := ABS(yRobotActual - yNode[i]);
	 diff_total[i] := diff_x[i] + diff_y[i];
 END_FOR
 
 min_total := 1000000;
 
 FOR m := 1 TO 170 BY 1 DO
	 IF min_total >= diff_total[m] THEN
		 min_total := diff_total[m];
		 startNode := m;
	 END_IF
 END_FOR
 
 /////////////////////////////////////////////////////AStern Algorithmus////////////////////////////////////////////////////////////////////////////////
 currentNode := startNode;
 h := SQRT(EXPT(xNode[startNode]-xEnd,2) + EXPT(yNode[startNode]-yEnd,2));
 f := g + h;
 
 //insert start node in openList
 openList[1,1] := 1;
 openList[1,2] := startNode;
 openList[1,3] := g;
 openList[1,4] := h;
 openList[1,5] := f;
 openList[1,6] := parentNode;
 
 //put in closedList
 closedList[1] := startNode;
 openList[1,1] := 0;
 
 //Goal reached?
 WHILE currentNode <> endNode AND NOT AStarFailed DO
	 //clear neighborlist
 	countNeighbor := 1;
	neighborList := nullMatrix_Neighbor;
	
	//search the neightbor and put in neighborlist
	FOR v := 1 TO 170 BY 1 DO
		//calculate forwards
		IF matrix[currentNode,v] <> 0 THEN
			g := gprev + SQRT(EXPT(xNode[v]-xNode[currentNode],2) + EXPT(yNode[v]-yNode[currentNode],2));
			h := SQRT(EXPT(xNode[v]-xEnd,2) + EXPT(yNode[v]-yEnd,2));
			neighborList[countNeighbor,1] := v;
			neighborList[countNeighbor,2] := g;
			neighborList[countNeighbor,3] := h;
			neighborList[countNeighbor,4] := g + h;
			neighborList[countNeighbor,5] := currentNode;
			countNeighbor := countNeighbor + 1;
		END_IF
	END_FOR
	
	IF countNeighbor = 1 THEN
		AStarFailed := TRUE;
	END_IF
	
	//possible neighbors will be inserted in openList
	FOR w := 1 TO 8 BY 1 DO
		flag := 0;
		FOR a := 1 TO 170 BY 1 DO
			//if already exist, update g, h, g and parent
			IF neighborList[w,1] = openList[a,2] THEN
				openList[a,5] := MIN(openList[a,5], neighborList[w,4]);
				IF openList[a,5] = neighborList[w,4] THEN
					openList[a,3] := neighborList[w,2];
					openList[a,4] := neighborList[w,3];
					openList[a,6] := neighborList[w,5];
				END_IF
				flag := 1;
			END_IF
		END_FOR
		IF flag = 0 AND neighborList[w,1] <> 0 THEN
			countOpen := countOpen +1;
			openList[countOpen,1] := 1;
			openList[countOpen,2] := neighborList[w,1]; //node
			openList[countOpen,3] := neighborList[w,2]; //g
			openList[countOpen,4] := neighborList[w,3]; //h
			openList[countOpen,5] := neighborList[w,4]; //f
			openList[countOpen,6] := neighborList[w,5]; //parent
		END_IF
	END_FOR
	 
	//find out the node with the smallest fn
	countTemp := 1;
	tempArray := nullMatrix_TempArray;
	FOR b := 1 TO countOpen BY 1 DO
		IF openList[b,1] = 1 THEN
			tempArray[countTemp, 1] := openList[b, 1];
			tempArray[countTemp, 2] := openList[b, 2];
			tempArray[countTemp, 3] := openList[b, 3];
			tempArray[countTemp, 4] := openList[b, 4];
			tempArray[countTemp, 5] := openList[b, 5];
			tempArray[countTemp, 6] := openList[b, 6];
			tempArray[countTemp, 7] := b;
			countTemp := countTemp + 1;
		END_IF
	END_FOR
	FOR d := 1 TO 170 BY 1 DO
		IF tempArray[d,5] = 0 THEN
			tempArray[d,5] := 10000000;
		END_IF
	END_FOR
	
	minf := 100000;
	
	FOR e := 1 TO 170 BY 1 DO
		IF tempArray[e,5] < minf THEN
			minf := tempArray[e,5];
			indexMin := LREAL_TO_INT(tempArray[e,7]);
		END_IF
	END_FOR
	
	//found smallest fn, update openList and put in closedList
	openList[indexMin, 1] := 0;
	currentNode := LREAL_TO_INT(openList[indexMin, 2]);
	gprev := openList[indexMin,3];
	countClosed := countClosed + 1;
	closedList[countClosed] := currentNode;
	
	IF currentNode = 0 OR countClosed > 170 OR countOpen > 170 THEN
		AStarFailed := TRUE;
	END_IF
 END_WHILE
 
 //Optimal path is generated by starting of the goal node to start node
 FOR k := countClosed TO 1 BY -1 DO
	 IF currentNode <> startNode THEN
		 wayPointList[countPointList] := currentNode;
		 FOR p := 1 TO countOpen BY 1 DO
			 IF openList[p,2] = currentNode THEN
				 currentNode := LREAL_TO_INT(openList[p,6]);
			 END_IF
		 END_FOR
		 countPointList := countPointList + 1;
	 ELSE
		wayPointList[countPointList] := currentNode;
		EXIT;
	 END_IF
 END_FOR

 FOR c := countPointList TO 1 BY -1 DO
	 wayPointList_finished[q] := wayPointList[c];
	 q := q + 1;
 END_FOR
 
 //////////////////////////////////////////////////Liste in Koordinaten/////////////////////////////////////////////////
 
//WayPointList in Koordinaten umwandeln
FOR t := 0 TO 100 BY 1 DO
	IF wayPointList_finished[t] <> 0 THEN
		xCoordinates[t] := xNode[wayPointList_finished[t]];
		yCoordinates[t] := yNode[wayPointList_finished[t]];
	END_IF
END_FOR
 
 IF NOT AStarFailed THEN
	 finishedASearch := TRUE;
 END_IF

METHOD reset : BOOL
VAR_INPUT
END_VAR

VAR
	numb: INT;
END_VAR
Zeros_INT(wayPointList_finished);
Zeros(closedList);
zeros_INT(wayPointList);
zeros(xCoordinates);
zeros(yCoordinates);
zeros(xNode);
zeros(yNode);
zeros(diff_x);
zeros(diff_y);
zeros(diff_total);

finishedASearch := FALSE;
numberOfNodes := 144;
q := 0;
numberOfColumns := 18;
parentNode := 0;
g := 0;
gprev := 0;
flag := FALSE;
countOpen := 1;
countTemp := 1;
countClosed := 1;
countPointList := 1;
AStarFailed := FALSE;

FOR numb := 16 TO 30 BY 1 DO
	removeNode[numb] := 0;
END_FOR
END_METHOD

END_FUNCTION_BLOCK

// ---- POUs/UserPOUs/UserFunctions/ZEROS_INT.TcPOU
//Fills an array of LREAL of varible length with zeros
FUNCTION ZEROS_INT
VAR_IN_OUT
	arr: ARRAY [*] OF INT;
END_VAR
VAR
	i : DINT := 0;
END_VAR

FOR i := LOWER_BOUND(arr,1) TO UPPER_BOUND(arr, 1) BY 1 DO
	arr[i] := 0;
END_FOR

END_FUNCTION

// ---- POUs/UserPOUs/GW2/ReadAssigment.TcPOU
FUNCTION_BLOCK ReadAssigment
VAR_INPUT
	assigment : Auftrag;
END_VAR
VAR_OUTPUT
	pointsFromSlotToReader : ARRAY[0..100] OF RobotPoseSimple;	//Weg vom Abholort zur Abmeldung 
	pointsFromReaderToSlot : ARRAY[0..100] OF RobotPoseSimple;	//Weg vom Abmelden zur Ablage
	lastPointsToCharging : ARRAY[0..2] OF RobotPoseSimple; 		//letzte Wegpunkte zur Ladestation
	lastNodePickUp, lastNodeStorage, pickupLocation, readerCheckOut, readerCheckIn, storageLocation, lastNodeCharging, chargingLocation : RobotPoseSimple;
	parkingSlots : ARRAY[1..4] OF RobotPoseSimple;				//Array mit Parkplätzen der Roboter
	endNodePickup, endNodeStorage, endNodeCharging : INT;		//Endknoten
	endNodeParking : ARRAY[1..4] OF INT;						//Knoten für Parkplätze
END_VAR
VAR
END_VAR

//FB zur Verarbeitung der Daten, die aus dem Auftrag kommen
//es werden Wegpunkte zum Anhängen an die Wegpunktliste und auch Wegpunktlisten zur An- und Abmeldung am RFID Reader generiert

IF assigment.Art = 'Fahrauftrag' THEN
	//////////////////////////////////////////////////////////////////////////////////////////////////////////////
	//////////////////////////////////FAHRAUFTRAG/////////////////////////////////////////////////////////////////
	//////////////////////////////////////////////////////////////////////////////////////////////////////////////
	
	//Abholort auswerten
	IF assigment.AbholStation = 1 THEN
		IF assigment.AbholTasche = 1 THEN
			//RFID links anfahren
			lastNodePickUp := ToRobotPoseSimple(x := 790, y := 2838, theta := -1);
			pickupLocation := ToRobotPoseSimple(x := 900, y := 2838, theta := 0); 
			readerCheckOut := ToRobotPoseSimple(x := 900, y := 2936, theta := 0); 
			endNodePickup := 146;
		ELSIF assigment.AbholTasche = 2 THEN
			//RFID links anfahren
			lastNodePickUp := ToRobotPoseSimple(x := 790, y := 2735, theta := -1);
			pickupLocation := ToRobotPoseSimple(x := 900, y := 2735, theta := 0); 
			readerCheckOut := ToRobotPoseSimple(x := 900, y := 2936, theta := 0); 
			endNodePickup := 145;
		ELSIF assigment.AbholTasche = 3 THEN
			//RFID rechts anfahren
			lastNodePickUp := ToRobotPoseSimple(x := 1410, y := 2835, theta := -1);
			pickupLocation := ToRobotPoseSimple(x := 1303, y := 2835, theta := pi); 
			readerCheckOut := ToRobotPoseSimple(x := 1303, y := 2935, theta := pi);	
			endNodePickup := 149;
		ELSIF assigment.AbholTasche = 4 THEN
			//RFID rechts anfahren	
			lastNodePickUp := ToRobotPoseSimple(x := 1410, y := 2736, theta := -1);
			pickupLocation := ToRobotPoseSimple(x := 1300, y := 2736, theta := pi);	
			readerCheckOut := ToRobotPoseSimple(x := 1303, y := 2935, theta := pi);	
			endNodePickup := 148;			
		END_IF
	ELSIF assigment.AbholStation = 2 THEN
		IF assigment.AbholTasche = 1 THEN
			//RFID links anfahren
			lastNodePickUp := ToRobotPoseSimple(x := 1990, y := 2829, theta := -1);
			pickupLocation := ToRobotPoseSimple(x := 2100, y := 2829, theta := 0); 
			readerCheckOut := ToRobotPoseSimple(x := 2110, y := 2931, theta := 0);
			endNodePickup := 152;
		ELSIF assigment.AbholTasche = 2 THEN
			//RFID links anfahren
			lastNodePickUp := ToRobotPoseSimple(x := 1990, y := 2731, theta := -1);
			pickupLocation := ToRobotPoseSimple(x := 2110, y := 2731, theta := 0); 
			readerCheckOut := ToRobotPoseSimple(x := 2110, y := 2931, theta := 0);
			endNodePickup := 151;
		ELSIF assigment.AbholTasche = 3 THEN
			//RFID rechts anfahren
			lastNodePickUp := ToRobotPoseSimple(x := 2550, y := 2833, theta := -1);
			pickupLocation := ToRobotPoseSimple(x := 2435, y := 2833, theta := pi);	
			readerCheckOut := ToRobotPoseSimple(x := 2435, y := 2940, theta := pi);	
			endNodePickup := 155;	
		ELSIF assigment.AbholTasche = 4 THEN
			//RFID rechts anfahren
			lastNodePickUp := ToRobotPoseSimple(x := 2550, y := 2732, theta := -1);
			pickupLocation := ToRobotPoseSimple(x := 2435, y := 2732, theta := pi);	
			readerCheckOut := ToRobotPoseSimple(x := 2435, y := 2940, theta := pi);	
			endNodePickup := 154;			
		END_IF
	ELSIF assigment.AbholStation = 3 THEN
		IF assigment.AbholTasche = 1 THEN
			//RFID links anfahren
			lastNodePickUp := ToRobotPoseSimple(x := 3130, y := 2837, theta := -1);
			pickupLocation := ToRobotPoseSimple(x := 3244, y := 2837, theta := 0);
			readerCheckOut := ToRobotPoseSimple(x := 3244, y := 2940, theta := 0);
			endNodePickup := 158;
		ELSIF assigment.AbholTasche = 2 THEN
			//RFID links anfahren
			lastNodePickUp := ToRobotPoseSimple(x := 3130, y := 2732, theta := -1);
			pickupLocation := ToRobotPoseSimple(x := 3244, y := 2732, theta := 0);
			readerCheckOut := ToRobotPoseSimple(x := 3244, y := 2940, theta := 0);
			endNodePickup := 157;
		ELSIF assigment.AbholTasche = 3 THEN
			//RFID rechts anfahren
			lastNodePickUp := ToRobotPoseSimple(x := 3760, y := 2840, theta := -1);
			pickupLocation := ToRobotPoseSimple(x := 3643, y := 2840, theta := pi); 
			readerCheckOut := ToRobotPoseSimple(x := 3662, y := 2940, theta := pi); 
			endNodePickup := 161;	
		ELSIF assigment.AbholTasche = 4 THEN
			//RFID rechts anfahren
			lastNodePickUp := ToRobotPoseSimple(x := 3760, y := 2732, theta := -1);
			pickupLocation := ToRobotPoseSimple(x := 3640, y := 2732, theta := pi);
			readerCheckOut := ToRobotPoseSimple(x := 3662, y := 2940, theta := pi);
			endNodePickup := 160;			
		END_IF
	ELSIF assigment.AbholStation = 4 THEN
		IF assigment.AbholTasche = 1 THEN
			//RFID links anfahren
			lastNodePickUp := ToRobotPoseSimple(x := 4360, y := 2838, theta := -1);
			pickupLocation := ToRobotPoseSimple(x := 4470, y := 2838, theta := 0); 
			readerCheckOut := ToRobotPoseSimple(x := 4470, y := 2940, theta := 0); 
			endNodePickup := 164;
		ELSIF assigment.AbholTasche = 2 THEN
			//RFID links anfahren
			lastNodePickUp := ToRobotPoseSimple(x := 4360, y := 2732, theta := -1);
			pickupLocation := ToRobotPoseSimple(x := 4470, y := 2732, theta := 0);
			readerCheckOut := ToRobotPoseSimple(x := 4470, y := 2940, theta := 0);
			endNodePickup := 163;
		ELSIF assigment.AbholTasche = 3 THEN
			//RFID rechts anfahren
			lastNodePickUp := ToRobotPoseSimple(x := 5000, y := 2855, theta := -1);
			pickupLocation := ToRobotPoseSimple(x := 4875, y := 2855, theta := pi); 
			readerCheckOut := ToRobotPoseSimple(x := 4875, y := 2942, theta := pi);	
			endNodePickup := 167;
		ELSIF assigment.AbholTasche = 4 THEN
			//RFID rechts anfahren
			lastNodePickUp := ToRobotPoseSimple(x := 5000, y := 2737, theta := -1);
			pickupLocation := ToRobotPoseSimple(x := 4870, y := 2737, theta := pi); 
			readerCheckOut := ToRobotPoseSimple(x := 4875, y := 2942, theta := pi);	
			endNodePickup := 166;			
		END_IF	
	END_IF
	

	//Ablageort auswerten
	IF assigment.AblageStation = 1 THEN
		IF assigment.AblageTasche = 1 THEN
			//RFID links anfahren
			lastNodeStorage := ToRobotPoseSimple(x := 790, y := 2838, theta := -1); 
			storageLocation := ToRobotPoseSimple(x := 900, y := 2838, theta := 0);
			readerCheckIn := ToRobotPoseSimple(x := 900, y := 2936, theta := 0);
			endNodeStorage := 147;
		ELSIF assigment.AblageTasche = 2 THEN
			//RFID links anfahren
			lastNodeStorage := ToRobotPoseSimple(x := 790, y := 2735, theta := -1); 
			storageLocation := ToRobotPoseSimple(x := 900, y := 2735, theta := 0);
			readerCheckIn := ToRobotPoseSimple(x := 900, y := 2936, theta := 0); 
			endNodeStorage := 147;
		ELSIF assigment.AblageTasche = 3 THEN
			//RFID rechts anfahren	
			lastNodeStorage := ToRobotPoseSimple(x := 1410, y := 2835, theta := -1);
			storageLocation := ToRobotPoseSimple(x := 1303, y := 2835, theta := pi);
			readerCheckIn := ToRobotPoseSimple(x := 1303, y := 2935, theta := pi);	
			endNodeStorage := 150;
		ELSIF assigment.AblageTasche = 4 THEN
			//RFID rechts anfahren	
			lastNodeStorage := ToRobotPoseSimple(x := 1410, y := 2736, theta := -1);
			storageLocation := ToRobotPoseSimple(x := 1300, y := 2736, theta := pi);
			readerCheckIn := ToRobotPoseSimple(x := 1303, y := 2935, theta := pi);
			endNodeStorage := 150;		
		END_IF
	ELSIF assigment.AblageStation = 2 THEN
		IF assigment.AblageTasche = 1 THEN
			//RFID links anfahren
			lastNodeStorage := ToRobotPoseSimple(x := 1990, y := 2829, theta := -1);
			storageLocation := ToRobotPoseSimple(x := 2100, y := 2829, theta := 0);
			readerCheckIn := ToRobotPoseSimple(x := 2105, y := 2931, theta := 0);
			endNodeStorage := 153;
		ELSIF assigment.AblageTasche = 2 THEN
			//RFID links anfahren
			lastNodeStorage := ToRobotPoseSimple(x := 1990, y := 2731, theta := -1);
			storageLocation := ToRobotPoseSimple(x := 2110, y := 2731, theta := 0);	
			readerCheckIn := ToRobotPoseSimple(x := 2110, y := 2931, theta := 0); 
			endNodeStorage := 153;
		ELSIF assigment.AblageTasche = 3 THEN
			//RFID rechts anfahren	
			lastNodeStorage := ToRobotPoseSimple(x := 2550, y := 2833, theta := -1);
			storageLocation := ToRobotPoseSimple(x := 2435, y := 2833, theta := pi);
			readerCheckIn := ToRobotPoseSimple(x := 2435, y := 2940, theta := pi);	
			endNodeStorage := 156;
		ELSIF assigment.AblageTasche = 4 THEN
			//RFID rechts anfahren	
			lastNodeStorage := ToRobotPoseSimple(x := 2550, y := 2732, theta := -1);
			storageLocation := ToRobotPoseSimple(x := 2435, y := 2732, theta := pi);
			readerCheckIn := ToRobotPoseSimple(x := 2435, y := 2940, theta := pi);
			endNodeStorage := 156;			
		END_IF
	ELSIF assigment.AblageStation = 3 THEN
		IF assigment.AblageTasche = 1 THEN
			//RFID links anfahren
			lastNodeStorage := ToRobotPoseSimple(x := 3130, y := 2837, theta := -1);
			storageLocation := ToRobotPoseSimple(x := 3244, y := 2837, theta := 0); 
			readerCheckIn := ToRobotPoseSimple(x := 3244, y := 2940, theta := 0);
			endNodeStorage := 159;
		ELSIF assigment.AblageTasche = 2 THEN
			//RFID links anfahren
			lastNodeStorage := ToRobotPoseSimple(x := 3130, y := 2732, theta := -1);
			storageLocation := ToRobotPoseSimple(x := 3244, y := 2732, theta := 0);
			readerCheckIn := ToRobotPoseSimple(x := 3244, y := 2940, theta := 0);
			endNodeStorage := 159;
		ELSIF assigment.AblageTasche = 3 THEN
			//RFID rechts anfahren
			lastNodeStorage := ToRobotPoseSimple(x := 3760, y := 2840, theta := -1);
			storageLocation := ToRobotPoseSimple(x := 3643, y := 2840, theta := pi);
			readerCheckIn := ToRobotPoseSimple(x := 3662, y := 2940, theta := pi);	
			endNodeStorage := 162;	
		ELSIF assigment.AblageTasche = 4 THEN
			//RFID rechts anfahren	
			lastNodeStorage := ToRobotPoseSimple(x := 3760, y := 2732, theta := -1);
			storageLocation := ToRobotPoseSimple(x := 3640, y := 2732, theta := pi);
			readerCheckIn := ToRobotPoseSimple(x := 3652, y := 2940, theta := pi);	
			endNodeStorage := 162;	
		END_IF
	ELSIF assigment.AblageStation = 4 THEN
		IF assigment.AblageTasche = 1 THEN
			//RFID links anfahren
			lastNodeStorage := ToRobotPoseSimple(x := 4360, y := 2838, theta := -1);
			storageLocation := ToRobotPoseSimple(x := 4470, y := 2838, theta := 0);
			readerCheckIn := ToRobotPoseSimple(x := 4470, y := 2940, theta := 0);
			endNodeStorage := 165;
		ELSIF assigment.AblageTasche = 2 THEN
			//RFID links anfahren
			lastNodeStorage := ToRobotPoseSimple(x := 4360, y := 2732, theta := -1);
			storageLocation := ToRobotPoseSimple(x := 4470, y := 2732, theta := 0);
			readerCheckIn := ToRobotPoseSimple(x := 4470, y := 2940, theta := 0);
			endNodeStorage := 165;
		ELSIF assigment.AblageTasche = 3 THEN
			//RFID rechts anfahren	
			lastNodeStorage := ToRobotPoseSimple(x := 5000, y := 2844, theta := -1);
			storageLocation := ToRobotPoseSimple(x := 4875, y := 2844, theta := pi);
			readerCheckIn := ToRobotPoseSimple(x := 4875, y := 2934, theta := pi);
			endNodeStorage := 168;
		ELSIF assigment.AblageTasche = 4 THEN
			//RFID rechts anfahren	
			lastNodeStorage := ToRobotPoseSimple(x := 5000, y := 2737, theta := -1);
			storageLocation := ToRobotPoseSimple(x := 4870, y := 2737, theta := pi);
			readerCheckIn := ToRobotPoseSimple(x := 4875, y := 2934, theta := pi);
			endNodeStorage := 168;		
		END_IF		
	END_IF
	
	//3 Wegpunkte für Fahrt von Tasche zu RFID Leser
	pointsFromSlotToReader[0] := pickupLocation;
	pointsFromSlotToReader[1] := ToRobotPoseSimple(x := lastNodePickUp.x, y := pickupLocation.y, theta := pickupLocation.theta);
	pointsFromSlotToReader[2] := ToRobotPoseSimple(x := lastNodePickUp.x, y := readerCheckOut.y, theta := readerCheckOut.theta);
	pointsFromSlotToReader[3] := readerCheckOut;
	pointsFromSlotToReader[4] := ToRobotPoseSimple(x := -1, y := -1, theta := -1);
	
	//3 Wegpunkte von RFID Leser zu Ablagetasche
	pointsFromReaderToSlot[0] := readerCheckIn;
	pointsFromReaderToSlot[1] := ToRobotPoseSimple(x := lastNodeStorage.x, y := readerCheckIn.y, theta := readerCheckIn.theta);
	pointsFromReaderToSlot[2] := ToRobotPoseSimple(x := lastNodeStorage.x, y := storageLocation.y, theta := storageLocation.theta);
	pointsFromReaderToSlot[3] := storageLocation;
	pointsFromReaderToSlot[4] := ToRobotPoseSimple(x := -1, y := -1, theta := -1);

	
ELSIF assigment.Art = 'Ladeauftrag' THEN
//////////////////////////////////////////////////////////////////////////////////////////////////////////////
///////////////////////////////////////LADEAUFTRAG////////////////////////////////////////////////////////////
//////////////////////////////////////////////////////////////////////////////////////////////////////////////

//Abholstation gibt an ob Ladestation 1 oder 2, Rest der Werte wird ignoriert	
	IF assigment.AbholStation = 1 THEN
		lastNodeCharging := ToRobotPoseSimple(x := 6117, y := 3100, theta := -1);
		chargingLocation := ToRobotPoseSimple(x := 6117, y := 3500, theta := 15.2*pi/180);
		endNodeCharging := 169;
	ELSIF assigment.AbholStation = 2 THEN
		lastNodeCharging := ToRobotPoseSimple(x := 6716, y := 3100, theta := -1);
		chargingLocation := ToRobotPoseSimple(x := 6716, y := 3504, theta := 15.2*pi/180);
		endNodeCharging := 170;
	END_IF
	
	lastPointsToCharging[0] := chargingLocation;
	lastPointsToCharging[1] := ToRobotPoseSimple(x := -1, y := -1, theta := -1);
END_IF


//////////////////////////////////////////////////////////////////////////////////////////////////////////////
//////////////////////////////////Parkplätze/////////////////////////////////////////////////////////////////
//////////////////////////////////////////////////////////////////////////////////////////////////////////////

parkingSlots[1] := ToRobotPoseSimple(x := 1000, y := 500, theta := -1);
endNodeParking[1] := 3;
parkingSlots[2] := ToRobotPoseSimple(x := 2200, y := 500, theta := -1);
endNodeParking[2] := 6;
parkingSlots[3] := ToRobotPoseSimple(x := 3400, y := 500, theta := -1);
endNodeParking[3] := 9;
parkingSlots[4] := ToRobotPoseSimple(x := 4600, y := 500, theta := -1);
endNodeParking[4] := 12;

END_FUNCTION_BLOCK

